// TIA Portal project "PTAR" (V16)

(* hardware
DEVICE "S7-1200 station_1"  S7-1200 Station
   slot 0: "Rack_0"  S7-1200 Rack  Rack  V1.0
   slot 1: "PLC_1 Agua de servicio"  CPU 1214C DC/DC/Rly  6ES7 214-1HG40-0XB0  V4.4
   slot 2: "DI 16x24VDC/DQ 16xRelay_1"  SM 1223 DI16/DQ16 x relay  6ES7 223-1PL32-0XB0  V2.0
   slot 3: "DI 16x24VDC_1"  6ES7 221-1BH32-0XB0  V2.0
   slot 4: "DI 16x24VDC_2"  6ES7 221-1BH32-0XB0  V2.0
   slot 5: "DI 16x24VDC_3"  6ES7 221-1BH32-0XB0  V2.0
   slot 6: "AI 8x13BIT_1"  6ES7 231-4HF32-0XB0  V2.1
   slot 7: "AI 8x13BIT_2"  6ES7 231-4HF32-0XB0  V2.1
   slot 101: "CM 1241 (RS422/485)_1"  6ES7 241-1CH32-0XB0  V2.2
DEVICE "S7-1200 station_2"  S7-1200 Station
   slot 0: "Rack_0"  S7-1200 Rack  Rack  V1.0
   slot 1: "PLC_2 Compresores y agua potable"  CPU 1214C AC/DC/Rly  6ES7 214-1BG40-0XB0  V4.4
   slot 2: "DI 16x24VDC/DQ 16xRelay_1"  6ES7 223-1BL32-0XB0  V2.0
   slot 3: "DI 16x24VDC/DQ 16xRelay_2"  SM 1223 DI16/DQ16 x relay  6ES7 223-1PL32-0XB0  V2.0
   slot 4: "DI 16x24VDC_1"  6ES7 221-1BH32-0XB0  V2.0
   slot 5: "DI 16x24VDC_2"  6ES7 221-1BH32-0XB0  V2.0
   slot 6: "AI 8x13BIT_1"  6ES7 231-4HF32-0XB0  V2.1
   slot 7: "AI 8x13BIT_2"  6ES7 231-4HF32-0XB0  V2.1
   slot 101: "CM 1241 (RS422/485)_1"  6ES7 241-1CH32-0XB0  V2.2
*)

// ===== PLC "PLC_1 Agua de servicio"  CPU 1214C DC/DC/Rly =====

VAR_GLOBAL   // PLC tag table "Tabla de variables estándar"
   "PARO EMERGENCIA TAB AGUA SERVICIO LOCAL" AT %I0.0 : Bool;
   "FALLA BREAKER TOTALIZADOR" AT %I0.1 : Bool;
   "FALLA BREAKER BOMBA 096P001A" AT %I0.2 : Bool;
   "FALLA BREAKER BOMBA 096P001B" AT %I0.3 : Bool;
   "FALLA BREAKER BOMBA 096P001C" AT %I0.4 : Bool;
   "FALLA BREAKER BOMBA 096P001D" AT %I0.5 : Bool;
   "FALLA BREAKER BOMBA 096P001E" AT %I0.6 : Bool;
   "FALLA BREAKER BOMBA 096P001F" AT %I0.7 : Bool;
   "SELEC TAB MODO CCM BOMBA 096P001A" AT %I1.0 : Bool;
   "SELEC TAB MODO CAMPO BOMBA 096P001A" AT %I1.1 : Bool;
   "SELEC TAB MODO REMOTO BOMBA 096P001A" AT %I1.2 : Bool;
   "SELEC TAB MODO CCM BOMBA 096P001B" AT %I1.3 : Bool;
   "SELEC TAB MODO CAMPO BOMBA 096P001B" AT %I1.4 : Bool;
   "SELEC TAB MODO REMOTO BOMBA 096P001B" AT %I1.5 : Bool;
   "SELEC TAB MODO CCM BOMBA 096P001C" AT %I2.0 : Bool;
   "SELEC TAB MODO CAMPO BOMBA 096P001C" AT %I2.1 : Bool;
   "SELEC TAB MODO REMOTO BOMBA 096P001C" AT %I2.2 : Bool;
   "SELEC TAB MODO CCM BOMBA 096P001D" AT %I2.3 : Bool;
   "SELEC TAB MODO CAMPO BOMBA 096P001D" AT %I2.4 : Bool;
   "SELEC TAB MODO REMOTO BOMBA 096P001D" AT %I2.5 : Bool;
   "SELEC TAB MODO CCM BOMBA 096P001E" AT %I2.6 : Bool;
   "SELEC TAB MODO CAMPO BOMBA 096P001E" AT %I2.7 : Bool;
   "SELEC TAB MODO REMOTO BOMBA 096P001E" AT %I3.0 : Bool;
   "SELEC TAB MODO CCM BOMBA 096P001F" AT %I3.1 : Bool;
   "SELEC TAB MODO CAMPO BOMBA 096P001F" AT %I3.2 : Bool;
   "SELEC TAB MODO REMOTO BOMBA 096P001F" AT %I3.3 : Bool;
   "PULSADOR START CCM 096P001A" AT %I3.4 : Bool;
   "PULSADOR STOP CCM 096P001A" AT %I3.5 : Bool;
   "PULSADOR START CCM 096P001B" AT %I3.6 : Bool;
   "PULSADOR STOP CCM 096P001B" AT %I3.7 : Bool;
   "PULSADOR START CCM 096P001C" AT %I4.0 : Bool;
   "PULSADOR STOP CCM 096P001C" AT %I4.1 : Bool;
   "PULSADOR START CCM 096P001D" AT %I4.2 : Bool;
   "PULSADOR STOP CCM 096P001D" AT %I4.3 : Bool;
   "PULSADOR START CCM 096P001E" AT %I4.4 : Bool;
   "PULSADOR STOP CCM 096P001E" AT %I4.5 : Bool;
   "PULSADOR START CCM 096P001F" AT %I4.6 : Bool;
   "PULSADOR STOP CCM 096P001F" AT %I4.7 : Bool;
   "PULSADOR RESET CCM 096P001A" AT %I5.0 : Bool;
   "PULSADOR RESET CCM 096P001B" AT %I5.1 : Bool;
   "PULSADOR RESET CCM 096P001C" AT %I5.2 : Bool;
   "PULSADOR RESET CCM 096P001D" AT %I5.3 : Bool;
   "PULSADOR RESET CCM 096P001E" AT %I5.4 : Bool;
   "PULSADOR RESET CCM 096P001F" AT %I5.5 : Bool;
   "PARO EMERGENCIA 096P001A CAMPO" AT %I7.5 : Bool;
   "PULSADOR START CAMPO 096P001A" AT %I5.7 : Bool;
   "PULSADOR STOP CAMPO 096P001A" AT %I6.0 : Bool;
   "PULSADOR START CAMPO 096P001B" AT %I6.1 : Bool;
   "PULSADOR STOP CAMPO 096P001B" AT %I6.2 : Bool;
   "PULSADOR START CAMPO 096P001C" AT %I6.3 : Bool;
   "PULSADOR STOP CAMPO 096P001C" AT %I6.4 : Bool;
   "PULSADOR START CAMPO 096P001D" AT %I6.5 : Bool;
   "PULSADOR STOP CAMPO 096P001D" AT %I6.6 : Bool;
   "PULSADOR START CAMPO 096P001E" AT %I6.7 : Bool;
   "PULSADOR STOP CAMPO 096P001E" AT %I7.0 : Bool;
   "PULSADOR START CAMPO 096P001F" AT %I7.1 : Bool;
   "PULSADOR STOP CAMPO 096P001F" AT %I7.2 : Bool;
   "SWITCH DE BAJA PRESION AGUA DE SERVICIO" AT %I7.3 : Bool;
   "SWITCH DE FLUJO AGUA DE SERVICIO" AT %I7.4 : Bool;
   "TRANSMISOR DE PRESION EN SUCCION 096PIT001" AT %IW300 : Word;
   "TRANSMISOR DE PRESION EN DESCARGA 096PIT002" AT %IW302 : Word;
   "PARO EMERGENCIA 096P001B CAMPO" AT %I7.6 : Bool;
   "PARO EMERGENCIA 096P001C CAMPO" AT %I7.7 : Bool;
   "PARO EMERGENCIA 096P001D CAMPO" AT %I8.0 : Bool;
   "PARO EMERGENCIA 096P001E CAMPO" AT %I8.1 : Bool;
   "PARO EMERGENCIA 096P001F CAMPO" AT %I8.2 : Bool;
   "PERMISO DE ARRANQUE" AT %I8.3 : Bool;
   "ENTRADAS DIGITALES GRUPO 1" AT %IW0 : Word;
   "ENTRADAS DIGITALES GRUPO 2" AT %IW2 : Word;
   "ENTRADAS DIGITALES GRUPO 3" AT %IW7 : Word;
   "Tag_1" AT %I8.4 : Bool;
   "OPERANDO BOMBA 096P001A" AT %Q0.0 : Bool;
   "FALLA BOMBA 096P001A" AT %Q0.1 : Bool;
   "OPERANDO BOMBA 096P001B" AT %Q0.2 : Bool;
   "FALLA BOMBA 096P001B" AT %Q0.3 : Bool;
   "OPERANDO BOMBA 096P001C" AT %Q0.4 : Bool;
   "FALLA BOMBA 096P001C" AT %Q0.5 : Bool;
   "OPERANDO BOMBA 096P001D" AT %Q0.6 : Bool;
   "FALLA BOMBA 096P001D" AT %Q0.7 : Bool;
   "OPERANDO BOMBA 096P001E" AT %Q1.0 : Bool;
   "FALLA BOMBA 096P001E" AT %Q1.1 : Bool;
   "OPERANDO BOMBA 096P001F" AT %Q2.0 : Bool;
   "FALLA BOMBA 096P001F" AT %Q2.1 : Bool;
   "SALIDAS DIGITALES GRUPO 1" AT %QW0 : Word;
   "CONSIGNA FRECUENCIA AGUA RESIDUAL" AT %MD100 : Real;
   "SLEEP BOOSTER" AT %M10.0 : Bool;
   "INICIAR BOMBA" AT %M10.1 : Bool;
   "Clock_Byte" AT %MB0 : Byte;
   "Clock_10Hz" AT %M0.0 : Bool;
   "Clock_5Hz" AT %M0.1 : Bool;
   "Clock_2.5Hz" AT %M0.2 : Bool;
   "Clock_2Hz" AT %M0.3 : Bool;
   "Clock_1.25Hz" AT %M0.4 : Bool;
   "Clock_1Hz" AT %M0.5 : Bool;
   "Clock_0.625Hz" AT %M0.6 : Bool;
   "Clock_0.5Hz" AT %M0.7 : Bool;
   "System_Byte" AT %MB1 : Byte;
   "FirstScan" AT %M1.0 : Bool;
   "DiagStatusUpdate" AT %M1.1 : Bool;
   "AlwaysTRUE" AT %M1.2 : Bool;
   "AlwaysFALSE" AT %M1.3 : Bool;
   "DISPONIBLE BOMBA A" AT %M10.2 : Bool;
   "DISPONIBLE BOMBA B" AT %M10.3 : Bool;
   "DISPONIBLE BOMBA C" AT %M10.4 : Bool;
   "DISPONIBLE BOMBA D" AT %M10.5 : Bool;
   "DISPONIBLE BOMBA E" AT %M10.6 : Bool;
   "DISPONIBLE BOMBA F" AT %M10.7 : Bool;
   "BOMBA LIDER 1" AT %M11.0 : Bool;
   "BOMBA LIDER 2" AT %M11.1 : Bool;
   "BOMBA LIDER 3" AT %M11.2 : Bool;
   "BOMBA LIDER 4" AT %M11.3 : Bool;
   "BOMBA LIDER 5" AT %M11.4 : Bool;
   "BOMBA LIDER 6" AT %M11.5 : Bool;
   "AD1" AT %M12.0 : Bool;
   "HABILITACION SISTEMA" AT %M12.1 : Bool;
   "AD2" AT %M12.2 : Bool;
   "AD3" AT %M12.3 : Bool;
   "AD4" AT %M12.4 : Bool;
   "AD5" AT %M12.5 : Bool;
   "ARRANQUE BOMBA A" AT %M13.0 : Bool;
   "ARRANQUE BOMBA B" AT %M13.1 : Bool;
   "ARRANQUE BOMBA C" AT %M13.2 : Bool;
   "ARRANQUE BOMBA D" AT %M13.4 : Bool;
   "ARRANQUE BOMBA E" AT %M13.5 : Bool;
   "ARRANQUE BOMBA F" AT %M13.6 : Bool;
   "PRESION OK" AT %M13.7 : Bool;
   "Tag_3" AT %M14.0 : Bool;
   "Tag_4" AT %M14.1 : Bool;
   "Tag_5" AT %M14.2 : Bool;
   "Tag_6" AT %M14.3 : Bool;
   "Tag_7" AT %M14.4 : Bool;
   "Tag_8" AT %M14.5 : Bool;
   "Tag_9" AT %M14.6 : Bool;
   "Tag_10" AT %M14.7 : Bool;
   "Tag_11" AT %M15.0 : Bool;
   "Tag_12" AT %M15.1 : Bool;
   "Tag_13" AT %M15.2 : Bool;
   "Tag_14" AT %M15.3 : Bool;
   "RESET GENERAL" AT %M2.0 : Bool;
   "ALARMA GENERAL" AT %M2.1 : Bool;
   "Tag_2" AT %M16.0 : Bool;
   "Tag_15" AT %M16.1 : Bool;
   "Tag_16" AT %M16.2 : Bool;
   "Tag_17" AT %M16.3 : Bool;
   "Tag_18" AT %M16.4 : Bool;
   "Tag_19" AT %M16.5 : Bool;
   "Tag_20" AT %M16.6 : Bool;
   "Tag_21" AT %M16.7 : Bool;
   "Tag_22" AT %M17.0 : Bool;
   "Tag_23" AT %M17.1 : Bool;
   "Tag_24" AT %M17.2 : Bool;
   "Tag_25" AT %M17.3 : Bool;
   "Tag_26" AT %M17.4 : Bool;
   "Tag_27" AT %M17.5 : Bool;
   "Tag_28" AT %M17.6 : Bool;
   "Tag_29" AT %M17.7 : Bool;
   "Tag_30" AT %M18.0 : Bool;
   "Tag_31" AT %M18.1 : Bool;
END_VAR

DATA_BLOCK "ANALOGAS"   // DB1
{ S7_Optimized_Access := 'TRUE' }
VERSION : 0.1
   VAR RETAIN
      "096PIT001" : Struct
         "CD MAX" : DInt := 27648;
         "CD MIN" : DInt := 0;
         "ING MAX" : Real := 232.0;
         "ING MIN" : Real := 0.0;
         HH : Real := 50.0;
         H : Real := 15.0;
         L : Real := 2.0;
         LL : Real := 1.5;
         ESCALIZADA : Real := 3.608217;
         PORCENTAJE : Real := 1.555266;
      END_STRUCT;
      "096PIT002" : Struct
         "CD MAX" : DInt := 27648;
         "CD MIN" : DInt := 0;
         "ING MAX" : Real := 232.0;
         "ING MIN" : Real := 0.0;
         HH : Real := 120.0;
         H : Real := 100.0;
         L : Real := 30.0;
         LL : Real := 20.0;
         ESCALIZADA : Real := 67.6331;
         PORCENTAJE : Real := 29.1522;
      END_STRUCT;
   END_VAR
BEGIN
END_DATA_BLOCK

DATA_BLOCK "BOTONERA"   // DB2
{ S7_Optimized_Access := 'TRUE' }
VERSION : 0.1
   VAR
      "096P001A" : Struct
         START : Bool;
         STOP : Bool;
         FALLA : Bool;
         "RESET FALLA" : Bool;
         "RESET TIEMPO OPERANDO" : Bool;
         "RESET TIEMPO ACUMULADO" : Bool;
      END_STRUCT;
      "096P001B" : Struct
         START : Bool;
         STOP : Bool;
         FALLA : Bool;
         "RESET FALLA" : Bool;
         "RESET TIEMPO OPERANDO" : Bool;
         "RESET TIEMPO ACUMULADO" : Bool;
      END_STRUCT;
      "096P001C" : Struct
         START : Bool;
         STOP : Bool;
         FALLA : Bool;
         "RESET FALLA" : Bool;
         "RESET TIEMPO OPERANDO" : Bool;
         "RESET TIEMPO ACUMULADO" : Bool;
      END_STRUCT;
      "096P001D" : Struct
         START : Bool;
         STOP : Bool;
         FALLA : Bool;
         "RESET FALLA" : Bool;
         "RESET TIEMPO OPERANDO" : Bool;
         "RESET TIEMPO ACUMULADO" : Bool;
      END_STRUCT;
      "096P001E" : Struct
         START : Bool;
         STOP : Bool;
         FALLA : Bool;
         "RESET FALLA" : Bool;
         "RESET TIEMPO OPERANDO" : Bool;
         "RESET TIEMPO ACUMULADO" : Bool;
      END_STRUCT;
      "096P001F" : Struct
         START : Bool;
         STOP : Bool;
         FALLA : Bool;
         "RESET FALLA" : Bool;
         "RESET TIEMPO OPERANDO" : Bool;
         "RESET TIEMPO ACUMULADO" : Bool;
      END_STRUCT;
      "TODO A MANUAL" : Bool;
      "TODO A AUTOMATICO" : Bool;
      "TODO EN MANUAL" : Bool;
      "TODO EN AUTOMATICO" : Bool;
   END_VAR
BEGIN
END_DATA_BLOCK

DATA_BLOCK "MODO OPERACION"   // DB3
{ S7_Optimized_Access := 'TRUE' }
VERSION : 0.1
   VAR RETAIN
      "096P001A" : Struct
         MANUAL : Bool;
         AUTOMATICO : Bool;
         SCADA : Bool;
      END_STRUCT;
      "096P001B" : Struct
         MANUAL : Bool;
         AUTOMATICO : Bool;
         SCADA : Bool;
      END_STRUCT;
      "096P001C" : Struct
         MANUAL : Bool;
         AUTOMATICO : Bool;
         SCADA : Bool;
      END_STRUCT;
      "096P001D" : Struct
         MANUAL : Bool;
         AUTOMATICO : Bool;
         SCADA : Bool;
      END_STRUCT;
      "096P001E" : Struct
         MANUAL : Bool;
         AUTOMATICO : Bool;
         SCADA : Bool;
      END_STRUCT;
      "096P001F" : Struct
         MANUAL : Bool;
         AUTOMATICO : Bool;
         SCADA : Bool;
      END_STRUCT;
   END_VAR
BEGIN
END_DATA_BLOCK

DATA_BLOCK "ESC HZ"   // DB4
{ S7_Optimized_Access := 'TRUE' }
VERSION : 0.1
   VAR RETAIN
      "096P001A" : Struct
         "FRECUENCIA MAX" : Real := 60.0;
         "FRECUENCIA MIN" : Real := 20.0;
         "FRECUENCIA OP" : Real := 60.0;
      END_STRUCT;
      "096P001B" : Struct
         "FRECUENCIA MAX" : Real := 60.0;
         "FRECUENCIA MIN" : Real := 20.0;
         "FRECUENCIA OP" : Real := 60.0;
      END_STRUCT;
      "096P001C" : Struct
         "FRECUENCIA MAX" : Real := 60.0;
         "FRECUENCIA MIN" : Real := 20.0;
         "FRECUENCIA OP" : Real := 60.0;
      END_STRUCT;
      "096P001D" : Struct
         "FRECUENCIA MAX" : Real := 60.0;
         "FRECUENCIA MIN" : Real := 20.0;
         "FRECUENCIA OP" : Real := 60.0;
      END_STRUCT;
      "096P001E" : Struct
         "FRECUENCIA MAX" : Real := 60.0;
         "FRECUENCIA MIN" : Real := 20.0;
         "FRECUENCIA OP" : Real := 60.0;
      END_STRUCT;
      "096P001F" : Struct
         "FRECUENCIA MAX" : Real := 60.0;
         "FRECUENCIA MIN" : Real := 20.0;
         "FRECUENCIA OP" : Real := 60.0;
      END_STRUCT;
   END_VAR
BEGIN
END_DATA_BLOCK

DATA_BLOCK "DATOS LECTURA VFDS"   // DB5
{ S7_Optimized_Access := 'TRUE' }
VERSION : 0.1
   VAR
      "096P001A" : Struct
         AMPERAJE : Real;
         FRECUENCIA : Real;
         "FRECUENCIA %" : Real;
         VOLTAJE : Real;
         ESTADO : Bool;
      END_STRUCT;
      "096P001B" : Struct
         AMPERAJE : Real;
         FRECUENCIA : Real;
         "FRECUENCIA %" : Real;
         VOLTAJE : Real;
         ESTADO : Bool;
      END_STRUCT;
      "096P001C" : Struct
         AMPERAJE : Real;
         FRECUENCIA : Real;
         "FRECUENCIA %" : Real;
         VOLTAJE : Real;
         ESTADO : Bool;
      END_STRUCT;
      "096P001D" : Struct
         AMPERAJE : Real;
         FRECUENCIA : Real;
         "FRECUENCIA %" : Real;
         VOLTAJE : Real;
         ESTADO : Bool;
      END_STRUCT;
      "096P001E" : Struct
         AMPERAJE : Real;
         FRECUENCIA : Real;
         "FRECUENCIA %" : Real;
         VOLTAJE : Real;
         ESTADO : Bool;
      END_STRUCT;
      "096P001F" : Struct
         AMPERAJE : Real;
         FRECUENCIA : Real;
         "FRECUENCIA %" : Real;
         VOLTAJE : Real;
         ESTADO : Bool;
      END_STRUCT;
   END_VAR
BEGIN
END_DATA_BLOCK

DATA_BLOCK "CONFIG SIS PRESION AGUA SERVICIO"   // DB25
{ S7_Optimized_Access := 'TRUE' }
VERSION : 0.1
   VAR RETAIN
      "DESVIO DE PRESION PARA DESPERTAR" : Real := 10.0;
      "VALOR DE FRECUENCIA PARA DORMIR" : Real := 40.0;
      "TIEMPO PARA MODO DORMIR" : Real := 40.0;
      "FRECUENCIA PARA ARRANCAR BOMBA EN PARALELO" : Real := 59.0;
      "TIEMPO PARA ARRANCAR BOMBA EN PARALELO" : Real := 40.0;
      "FRECUENCIA PARA APAGAR BOMBA EN PARALELO" : Real := 43.0;
      "TIEMPO PARA APAGAR BOMBA EN PARALELO" : Real := 5.0;
      "TORQUE MINIMO PARA DETECCION BOMBA EN VACIO" : Real := 20.0;
      "TIEMPO DETECCION BOMBA EN VACIO" : Real := 10.0;
      "PRESION BOOSTER" : Real := 2.0;
      "TIEMPO SLEEP BOOSTER" : Real := 10.0;
      "FRECUENCIA MAXIMA CONFIGURADA EN VFDS" : Real := 60.0;
      "FRECUENCIA MINIMA CONFIGURADA EN VFDS" : Real := 37.0;
      "TIEMPO DE ALTERNACION" : Int := 10;
      SETPOINT : Real := 80.0;
      "SETPOINT %" : Real := 34.61207;
      K : Real := 0.0;
      TI : Real := 0.0;
      TD : Real := 0.0;
   END_VAR
   VAR
      "SALIDA PID %" : Real := 0.0;
   END_VAR
BEGIN
END_DATA_BLOCK

DATA_BLOCK "DATOS ESCRITURA VFDS"   // DB30
{ S7_Optimized_Access := 'TRUE' }
VERSION : 0.1
   VAR
      "096P001A" : Struct
         FRECUENCIA : Real;
      END_STRUCT;
      "096P001B" : Struct
         FRECUENCIA : Real;
      END_STRUCT;
      "096P001C" : Struct
         FRECUENCIA : Real;
      END_STRUCT;
      "096P001D" : Struct
         FRECUENCIA : Real;
      END_STRUCT;
      "096P001E" : Struct
         FRECUENCIA : Real;
      END_STRUCT;
      "096P001F" : Struct
         FRECUENCIA : Real;
      END_STRUCT;
   END_VAR
BEGIN
END_DATA_BLOCK

DATA_BLOCK "Alarmas Sis servicio"   // DB37
{ S7_Optimized_Access := 'TRUE' }
VERSION : 0.1
   VAR
      "Alarma general" : Bool;
      "Reset alarmas" : Bool;
   END_VAR
BEGIN
END_DATA_BLOCK

DATA_BLOCK "LECTURA VFD1"   // DB40
{ S7_Optimized_Access := 'FALSE' }
VERSION : 0.1
   VAR
      "40007+" : Array[0..8] of Int;
      "40016+" : Array[0..7] of Int;
      "40816+" : Array[0..1] of Int;
   END_VAR
BEGIN
END_DATA_BLOCK

DATA_BLOCK "LECTURA VFD2"   // DB41
{ S7_Optimized_Access := 'FALSE' }
VERSION : 0.1
   VAR
      "40007+" : Array[0..8] of Int;
      "40016+" : Array[0..7] of Int;
      "40816+" : Array[0..1] of Int;
   END_VAR
BEGIN
END_DATA_BLOCK

DATA_BLOCK "LECTURA VFD3"   // DB42
{ S7_Optimized_Access := 'FALSE' }
VERSION : 0.1
   VAR
      "40007+" : Array[0..8] of Int;
      "40016+" : Array[0..7] of Int;
      "40816+" : Array[0..1] of Int;
   END_VAR
BEGIN
END_DATA_BLOCK

DATA_BLOCK "LECTURA VFD4"   // DB43
{ S7_Optimized_Access := 'FALSE' }
VERSION : 0.1
   VAR
      "40007+" : Array[0..8] of Int;
      "40016+" : Array[0..7] of Int;
      "40816+" : Array[0..1] of Int;
   END_VAR
BEGIN
END_DATA_BLOCK

DATA_BLOCK "LECTURA VFD5"   // DB44
{ S7_Optimized_Access := 'FALSE' }
VERSION : 0.1
   VAR
      "40007+" : Array[0..8] of Int;
      "40016+" : Array[0..7] of Int;
      "40816+" : Array[0..1] of Int;
   END_VAR
BEGIN
END_DATA_BLOCK

DATA_BLOCK "LECTURA VFD6"   // DB45
{ S7_Optimized_Access := 'FALSE' }
VERSION : 0.1
   VAR
      "40007+" : Array[0..8] of Int;
      "40016+" : Array[0..7] of Int;
      "40816+" : Array[0..1] of Int;
   END_VAR
BEGIN
END_DATA_BLOCK

DATA_BLOCK "ESCRITURA VFD1"   // DB47
{ S7_Optimized_Access := 'FALSE' }
VERSION : 0.1
   VAR
      "40005+" : Array[0..1] of Int;
   END_VAR
BEGIN
END_DATA_BLOCK

DATA_BLOCK "ESCRITURA VFD2"   // DB48
{ S7_Optimized_Access := 'FALSE' }
VERSION : 0.1
   VAR
      "40005+" : Array[0..1] of Int;
   END_VAR
BEGIN
END_DATA_BLOCK

DATA_BLOCK "ESCRITURA VFD3"   // DB49
{ S7_Optimized_Access := 'FALSE' }
VERSION : 0.1
   VAR
      "40005+" : Array[0..1] of Int;
   END_VAR
BEGIN
END_DATA_BLOCK

DATA_BLOCK "ESCRITURA VFD4"   // DB50
{ S7_Optimized_Access := 'FALSE' }
VERSION : 0.1
   VAR
      "40005+" : Array[0..1] of Int;
   END_VAR
BEGIN
END_DATA_BLOCK

DATA_BLOCK "ESCRITURA VFD5"   // DB51
{ S7_Optimized_Access := 'FALSE' }
VERSION : 0.1
   VAR
      "40005+" : Array[0..1] of Int;
   END_VAR
BEGIN
END_DATA_BLOCK

DATA_BLOCK "ESCRITURA VFD6"   // DB52
{ S7_Optimized_Access := 'FALSE' }
VERSION : 0.1
   VAR
      "40005+" : Array[0..1] of Int;
   END_VAR
BEGIN
END_DATA_BLOCK

DATA_BLOCK "DATA MODBUS TCP"   // DB78
{ S7_Optimized_Access := 'FALSE' }
VERSION : 0.1
   VAR
      DATA : Array[0..100] of Word;
   END_VAR
BEGIN
END_DATA_BLOCK

DATA_BLOCK "MB CONFIG"   // DB79
{ S7_Optimized_Access := 'FALSE' }
VERSION : 0.1
   VAR
      CONNECT : TCON_IP_v4;
      NDR : Bool;
      DR : Bool;
      ERROR : Bool;
      STATUS : Word;
   END_VAR
BEGIN
   CONNECT.InterfaceId := 64;
   CONNECT.ID := 1;
   CONNECT.ConnectionType := 11;
   CONNECT.LocalPort := 502;
END_DATA_BLOCK

DATA_BLOCK "FALLAS HMI"   // DB93
{ S7_Optimized_Access := 'FALSE' }
VERSION : 0.1
   VAR
      "PARO EMERGENCIA ACTIVO SISTEMA GRAL AGUA SERVICIO" : Bool;
      "FALLA BREAKER PRINCIPAL" : Bool;
      "FALLA BREAKER Q1 - VFD 1 096P001A" : Bool;
      "FALLA VARIADOR VELOCIDAD 096P001A" : Bool;
      "PARO DE EMERGENCIA ACTIVO 096P001A" : Bool;
      "NO CONFIRMA ARRANQUE BOMBA 096P001A" : Bool;
      "FALLA BREAKER Q2 - VFD 2 096P001B" : Bool;
      "FALLA VARIADOR VELOCIDAD 096P001B" : Bool;
      "PARO DE EMERGENCIA ACTIVO 096P001B" : Bool;
      "NO CONFIRMA ARRANQUE BOMBA 096P001B" : Bool;
      "FALLA BREAKER Q3 - VFD 3 096P001C" : Bool;
      "FALLA VARIADOR VELOCIDAD 096P001C" : Bool;
      "PARO DE EMERGENCIA ACTIVO 096P001C" : Bool;
      "NO CONFIRMA ARRANQUE BOMBA 096P001C" : Bool;
      "FALLA BREAKER Q4 - VFD 4 096P001D" : Bool;
      "FALLA VARIADOR VELOCIDAD 096P001D" : Bool;
      "PARO DE EMERGENCIA ACTIVO 096P001D" : Bool;
      "NO CONFIRMA ARRANQUE BOMBA 096P001D" : Bool;
      "FALLA BREAKER Q5 - VFD 5 096P001E" : Bool;
      "FALLA VARIADOR VELOCIDAD 096P001E" : Bool;
      "PARO DE EMERGENCIA ACTIVO 096P001E" : Bool;
      "NO CONFIRMA ARRANQUE BOMBA 096P001E" : Bool;
      "FALLA BREAKER Q6 - VFD 6 096P001F" : Bool;
      "FALLA VARIADOR VELOCIDAD 096P001F" : Bool;
      "PARO DE EMERGENCIA ACTIVO 096P001F" : Bool;
      "NO CONFIRMA ARRANQUE BOMBA 096P001F" : Bool;
      "SWITCH DE FLUJO EN SUCCION INACTIVO FSL001" : Bool;
      "SWITCH DE PRESION EN SUCCION INACTIVO PSL001" : Bool;
      "NO CONFIRMA SWITCH DE FLUJO CON BOMBA 096P001A" : Bool;
      "NO CONFIRMA SWITCH DE FLUJO CON BOMBA 096P001B" : Bool;
      "NO CONFIRMA SWITCH DE FLUJO CON BOMBA 096P001C" : Bool;
      "NO CONFIRMA SWITCH DE FLUJO CON BOMBA 096P001D" : Bool;
      "NO CONFIRMA SWITCH DE FLUJO CON BOMBA 096P001E" : Bool;
      "NO CONFIRMA SWITCH DE FLUJO CON BOMBA 096P001F" : Bool;
      "FALLA POR ALTA PRESION DE DESCARGA 096PIT002" : Bool;
      "ALARMA POR ALTA PRESION DE DESCARGA 096PIT002" : Bool;
      "ALARMA POR BAJA PRESION DE DESCARGA 096PIT002" : Bool;
      "FALLA POR BAJA PRESION DE DESCARGA 096PIT002" : Bool;
      "FALLA POR ALTA PRESION DE SUCCION 096PIT001" : Bool;
      "ALARMA POR ALTA PRESION DE SUCCION 096PIT001" : Bool;
      "ALARMA POR BAJA PRESION DE SUCCION 096PIT001" : Bool;
      "FALLA POR BAJA PRESION DE SUCCION 096PIT001" : Bool;
   END_VAR
BEGIN
END_DATA_BLOCK

// folder: System blocks/Program resources

DATA_BLOCK "TEMPO MODO MANUAL 001A"   // DB6
{ S7_Optimized_Access := 'TRUE' }
AUTHOR : Simatic
FAMILY : IEC
NAME : IEC_TMR
VERSION : 1.0
// stored: InstanceOfName IEC_TIMER
"IEC_TIMER"
BEGIN
END_DATA_BLOCK

DATA_BLOCK "TEMPO MODO AUTOMATICO 001A"   // DB7
{ S7_Optimized_Access := 'TRUE' }
AUTHOR : Simatic
FAMILY : IEC
NAME : IEC_TMR
VERSION : 1.0
// stored: InstanceOfName IEC_TIMER
"IEC_TIMER"
BEGIN
END_DATA_BLOCK

DATA_BLOCK "TEMPO MODO SCADA 001A"   // DB8
{ S7_Optimized_Access := 'TRUE' }
AUTHOR : Simatic
FAMILY : IEC
NAME : IEC_TMR
VERSION : 1.0
// stored: InstanceOfName IEC_TIMER
"IEC_TIMER"
BEGIN
END_DATA_BLOCK

DATA_BLOCK "TEMPO MODO MANUAL 001B"   // DB9
{ S7_Optimized_Access := 'TRUE' }
AUTHOR : Simatic
FAMILY : IEC
NAME : IEC_TMR
VERSION : 1.0
// stored: InstanceOfName IEC_TIMER
"IEC_TIMER"
BEGIN
END_DATA_BLOCK

DATA_BLOCK "TEMPO MODO AUTOMATICO 001B"   // DB10
{ S7_Optimized_Access := 'TRUE' }
AUTHOR : Simatic
FAMILY : IEC
NAME : IEC_TMR
VERSION : 1.0
// stored: InstanceOfName IEC_TIMER
"IEC_TIMER"
BEGIN
END_DATA_BLOCK

DATA_BLOCK "TEMPO MODO SCADA 001B"   // DB11
{ S7_Optimized_Access := 'TRUE' }
AUTHOR : Simatic
FAMILY : IEC
NAME : IEC_TMR
VERSION : 1.0
// stored: InstanceOfName IEC_TIMER
"IEC_TIMER"
BEGIN
END_DATA_BLOCK

DATA_BLOCK "TEMPO MODO MANUAL 001C"   // DB12
{ S7_Optimized_Access := 'TRUE' }
AUTHOR : Simatic
FAMILY : IEC
NAME : IEC_TMR
VERSION : 1.0
// stored: InstanceOfName IEC_TIMER
"IEC_TIMER"
BEGIN
END_DATA_BLOCK

DATA_BLOCK "TEMPO MODO AUTOMATICO 001C"   // DB13
{ S7_Optimized_Access := 'TRUE' }
AUTHOR : Simatic
FAMILY : IEC
NAME : IEC_TMR
VERSION : 1.0
// stored: InstanceOfName IEC_TIMER
"IEC_TIMER"
BEGIN
END_DATA_BLOCK

DATA_BLOCK "TEMPO MODO SCADA 001C"   // DB14
{ S7_Optimized_Access := 'TRUE' }
AUTHOR : Simatic
FAMILY : IEC
NAME : IEC_TMR
VERSION : 1.0
// stored: InstanceOfName IEC_TIMER
"IEC_TIMER"
BEGIN
END_DATA_BLOCK

DATA_BLOCK "TEMPO MODO MANUAL 001D"   // DB15
{ S7_Optimized_Access := 'TRUE' }
AUTHOR : Simatic
FAMILY : IEC
NAME : IEC_TMR
VERSION : 1.0
// stored: InstanceOfName IEC_TIMER
"IEC_TIMER"
BEGIN
END_DATA_BLOCK

DATA_BLOCK "TEMPO MODO AUTOMATICO 001D"   // DB16
{ S7_Optimized_Access := 'TRUE' }
AUTHOR : Simatic
FAMILY : IEC
NAME : IEC_TMR
VERSION : 1.0
// stored: InstanceOfName IEC_TIMER
"IEC_TIMER"
BEGIN
END_DATA_BLOCK

DATA_BLOCK "TEMPO MODO SCADA 001D"   // DB17
{ S7_Optimized_Access := 'TRUE' }
AUTHOR : Simatic
FAMILY : IEC
NAME : IEC_TMR
VERSION : 1.0
// stored: InstanceOfName IEC_TIMER
"IEC_TIMER"
BEGIN
END_DATA_BLOCK

DATA_BLOCK "TEMPO MODO MANUAL 001E"   // DB18
{ S7_Optimized_Access := 'TRUE' }
AUTHOR : Simatic
FAMILY : IEC
NAME : IEC_TMR
VERSION : 1.0
// stored: InstanceOfName IEC_TIMER
"IEC_TIMER"
BEGIN
END_DATA_BLOCK

DATA_BLOCK "TEMPO MODO AUTOMATICO 001E"   // DB19
{ S7_Optimized_Access := 'TRUE' }
AUTHOR : Simatic
FAMILY : IEC
NAME : IEC_TMR
VERSION : 1.0
// stored: InstanceOfName IEC_TIMER
"IEC_TIMER"
BEGIN
END_DATA_BLOCK

DATA_BLOCK "TEMPO MODO SCADA 001E"   // DB20
{ S7_Optimized_Access := 'TRUE' }
AUTHOR : Simatic
FAMILY : IEC
NAME : IEC_TMR
VERSION : 1.0
// stored: InstanceOfName IEC_TIMER
"IEC_TIMER"
BEGIN
END_DATA_BLOCK

DATA_BLOCK "TEMPO MODO SCADA 001F"   // DB21
{ S7_Optimized_Access := 'TRUE' }
AUTHOR : Simatic
FAMILY : IEC
NAME : IEC_TMR
VERSION : 1.0
// stored: InstanceOfName IEC_TIMER
"IEC_TIMER"
BEGIN
END_DATA_BLOCK

DATA_BLOCK "TEMPO MODO AUTOMATICO 001F"   // DB22
{ S7_Optimized_Access := 'TRUE' }
AUTHOR : Simatic
FAMILY : IEC
NAME : IEC_TMR
VERSION : 1.0
// stored: InstanceOfName IEC_TIMER
"IEC_TIMER"
BEGIN
END_DATA_BLOCK

DATA_BLOCK "TEMPO MODO MANUAL 001F"   // DB23
{ S7_Optimized_Access := 'TRUE' }
AUTHOR : Simatic
FAMILY : IEC
NAME : IEC_TMR
VERSION : 1.0
// stored: InstanceOfName IEC_TIMER
"IEC_TIMER"
BEGIN
END_DATA_BLOCK

DATA_BLOCK "TIEMPO PARA APAGAR"   // DB26
{ S7_Optimized_Access := 'TRUE' }
AUTHOR : Simatic
FAMILY : IEC
NAME : IEC_TMR
VERSION : 1.0
// stored: InstanceOfName IEC_TIMER
"IEC_TIMER"
BEGIN
END_DATA_BLOCK

DATA_BLOCK "TIEMPO SLEEP BOOSTER"   // DB27
{ S7_Optimized_Access := 'TRUE' }
AUTHOR : Simatic
FAMILY : IEC
NAME : IEC_TMR
VERSION : 1.0
// stored: InstanceOfName IEC_TIMER
"IEC_TIMER"
BEGIN
END_DATA_BLOCK

DATA_BLOCK "RESET SLEEP BOOSTER"   // DB28
{ S7_Optimized_Access := 'TRUE' }
AUTHOR : Simatic
FAMILY : IEC
NAME : IEC_TMR
VERSION : 1.0
// stored: InstanceOfName IEC_TIMER
"IEC_TIMER"
BEGIN
END_DATA_BLOCK

DATA_BLOCK "CONFIRMACION FLUJO 096P001A"   // DB31
{ S7_Optimized_Access := 'TRUE' }
AUTHOR : Simatic
FAMILY : IEC
NAME : IEC_TMR
VERSION : 1.0
// stored: InstanceOfName IEC_TIMER
"IEC_TIMER"
BEGIN
END_DATA_BLOCK

DATA_BLOCK "CONFIRMACION FLUJO 096P001B"   // DB32
{ S7_Optimized_Access := 'TRUE' }
AUTHOR : Simatic
FAMILY : IEC
NAME : IEC_TMR
VERSION : 1.0
// stored: InstanceOfName IEC_TIMER
"IEC_TIMER"
BEGIN
END_DATA_BLOCK

DATA_BLOCK "CONFIRMACION FLUJO 096P001C"   // DB33
{ S7_Optimized_Access := 'TRUE' }
AUTHOR : Simatic
FAMILY : IEC
NAME : IEC_TMR
VERSION : 1.0
// stored: InstanceOfName IEC_TIMER
"IEC_TIMER"
BEGIN
END_DATA_BLOCK

DATA_BLOCK "CONFIRMACION FLUJO 096P001D"   // DB34
{ S7_Optimized_Access := 'TRUE' }
AUTHOR : Simatic
FAMILY : IEC
NAME : IEC_TMR
VERSION : 1.0
// stored: InstanceOfName IEC_TIMER
"IEC_TIMER"
BEGIN
END_DATA_BLOCK

DATA_BLOCK "CONFIRMACION FLUJO 096P001E"   // DB35
{ S7_Optimized_Access := 'TRUE' }
AUTHOR : Simatic
FAMILY : IEC
NAME : IEC_TMR
VERSION : 1.0
// stored: InstanceOfName IEC_TIMER
"IEC_TIMER"
BEGIN
END_DATA_BLOCK

DATA_BLOCK "CONFIRMACION FLUJO 096P001F"   // DB36
{ S7_Optimized_Access := 'TRUE' }
AUTHOR : Simatic
FAMILY : IEC
NAME : IEC_TMR
VERSION : 1.0
// stored: InstanceOfName IEC_TIMER
"IEC_TIMER"
BEGIN
END_DATA_BLOCK

DATA_BLOCK "CONTADOR COMUNICACION"   // DB46
{ S7_Optimized_Access := 'TRUE' }
AUTHOR : Simatic
FAMILY : IEC
NAME : CNTR
VERSION : 1.0
// stored: InstanceOfName IEC_COUNTER
"IEC_COUNTER"
BEGIN
END_DATA_BLOCK

DATA_BLOCK "CONT SEG BA"   // DB53
{ S7_Optimized_Access := 'TRUE' }
AUTHOR : Simatic
FAMILY : IEC
NAME : CNTR
VERSION : 1.0
// stored: InstanceOfName IEC_COUNTER
"IEC_COUNTER"
BEGIN
END_DATA_BLOCK

DATA_BLOCK "CONT MIN BA"   // DB54
{ S7_Optimized_Access := 'TRUE' }
AUTHOR : Simatic
FAMILY : IEC
NAME : CNTR
VERSION : 1.0
// stored: InstanceOfName IEC_COUNTER
"IEC_COUNTER"
BEGIN
END_DATA_BLOCK

DATA_BLOCK "RESET BA"   // DB55
{ S7_Optimized_Access := 'TRUE' }
AUTHOR : Simatic
FAMILY : IEC
NAME : IEC_TMR
VERSION : 1.0
// stored: InstanceOfName IEC_TIMER
"IEC_TIMER"
BEGIN
END_DATA_BLOCK

DATA_BLOCK "CONT SEG BB"   // DB56
{ S7_Optimized_Access := 'TRUE' }
AUTHOR : Simatic
FAMILY : IEC
NAME : CNTR
VERSION : 1.0
// stored: InstanceOfName IEC_COUNTER
"IEC_COUNTER"
BEGIN
END_DATA_BLOCK

DATA_BLOCK "CONT MIN BB"   // DB57
{ S7_Optimized_Access := 'TRUE' }
AUTHOR : Simatic
FAMILY : IEC
NAME : CNTR
VERSION : 1.0
// stored: InstanceOfName IEC_COUNTER
"IEC_COUNTER"
BEGIN
END_DATA_BLOCK

DATA_BLOCK "RESET BB"   // DB58
{ S7_Optimized_Access := 'TRUE' }
AUTHOR : Simatic
FAMILY : IEC
NAME : IEC_TMR
VERSION : 1.0
// stored: InstanceOfName IEC_TIMER
"IEC_TIMER"
BEGIN
END_DATA_BLOCK

DATA_BLOCK "CONT SEG BC"   // DB59
{ S7_Optimized_Access := 'TRUE' }
AUTHOR : Simatic
FAMILY : IEC
NAME : CNTR
VERSION : 1.0
// stored: InstanceOfName IEC_COUNTER
"IEC_COUNTER"
BEGIN
END_DATA_BLOCK

DATA_BLOCK "CONT MIN BC"   // DB60
{ S7_Optimized_Access := 'TRUE' }
AUTHOR : Simatic
FAMILY : IEC
NAME : CNTR
VERSION : 1.0
// stored: InstanceOfName IEC_COUNTER
"IEC_COUNTER"
BEGIN
END_DATA_BLOCK

DATA_BLOCK "RESET BC"   // DB61
{ S7_Optimized_Access := 'TRUE' }
AUTHOR : Simatic
FAMILY : IEC
NAME : IEC_TMR
VERSION : 1.0
// stored: InstanceOfName IEC_TIMER
"IEC_TIMER"
BEGIN
END_DATA_BLOCK

DATA_BLOCK "CONT SEG BD"   // DB62
{ S7_Optimized_Access := 'TRUE' }
AUTHOR : Simatic
FAMILY : IEC
NAME : CNTR
VERSION : 1.0
// stored: InstanceOfName IEC_COUNTER
"IEC_COUNTER"
BEGIN
END_DATA_BLOCK

DATA_BLOCK "CONT MIN BD"   // DB63
{ S7_Optimized_Access := 'TRUE' }
AUTHOR : Simatic
FAMILY : IEC
NAME : CNTR
VERSION : 1.0
// stored: InstanceOfName IEC_COUNTER
"IEC_COUNTER"
BEGIN
END_DATA_BLOCK

DATA_BLOCK "RESET BD"   // DB64
{ S7_Optimized_Access := 'TRUE' }
AUTHOR : Simatic
FAMILY : IEC
NAME : IEC_TMR
VERSION : 1.0
// stored: InstanceOfName IEC_TIMER
"IEC_TIMER"
BEGIN
END_DATA_BLOCK

DATA_BLOCK "CONT SEG BE"   // DB65
{ S7_Optimized_Access := 'TRUE' }
AUTHOR : Simatic
FAMILY : IEC
NAME : CNTR
VERSION : 1.0
// stored: InstanceOfName IEC_COUNTER
"IEC_COUNTER"
BEGIN
END_DATA_BLOCK

DATA_BLOCK "CONT MIN BE"   // DB66
{ S7_Optimized_Access := 'TRUE' }
AUTHOR : Simatic
FAMILY : IEC
NAME : CNTR
VERSION : 1.0
// stored: InstanceOfName IEC_COUNTER
"IEC_COUNTER"
BEGIN
END_DATA_BLOCK

DATA_BLOCK "RESET BE"   // DB67
{ S7_Optimized_Access := 'TRUE' }
AUTHOR : Simatic
FAMILY : IEC
NAME : IEC_TMR
VERSION : 1.0
// stored: InstanceOfName IEC_TIMER
"IEC_TIMER"
BEGIN
END_DATA_BLOCK

DATA_BLOCK "CONT SEG BF"   // DB68
{ S7_Optimized_Access := 'TRUE' }
AUTHOR : Simatic
FAMILY : IEC
NAME : CNTR
VERSION : 1.0
// stored: InstanceOfName IEC_COUNTER
"IEC_COUNTER"
BEGIN
END_DATA_BLOCK

DATA_BLOCK "CONT MIN BF"   // DB69
{ S7_Optimized_Access := 'TRUE' }
AUTHOR : Simatic
FAMILY : IEC
NAME : CNTR
VERSION : 1.0
// stored: InstanceOfName IEC_COUNTER
"IEC_COUNTER"
BEGIN
END_DATA_BLOCK

DATA_BLOCK "RESET BF"   // DB70
{ S7_Optimized_Access := 'TRUE' }
AUTHOR : Simatic
FAMILY : IEC
NAME : IEC_TMR
VERSION : 1.0
// stored: InstanceOfName IEC_TIMER
"IEC_TIMER"
BEGIN
END_DATA_BLOCK

DATA_BLOCK "CONTADOR ALTERNACION"   // DB71
{ S7_Optimized_Access := 'TRUE' }
AUTHOR : Simatic
FAMILY : IEC
NAME : CNTR
VERSION : 1.0
// stored: InstanceOfName IEC_COUNTER
"IEC_COUNTER"
BEGIN
END_DATA_BLOCK

DATA_BLOCK "FALLA BOMBA LIDER 1"   // DB72
{ S7_Optimized_Access := 'TRUE' }
AUTHOR : Simatic
FAMILY : IEC
NAME : IEC_TMR
VERSION : 1.0
// stored: InstanceOfName IEC_TIMER
"IEC_TIMER"
BEGIN
END_DATA_BLOCK

DATA_BLOCK "FALLA BOMBA LIDER 6"   // DB73
{ S7_Optimized_Access := 'TRUE' }
AUTHOR : Simatic
FAMILY : IEC
NAME : IEC_TMR
VERSION : 1.0
// stored: InstanceOfName IEC_TIMER
"IEC_TIMER"
BEGIN
END_DATA_BLOCK

DATA_BLOCK "FALLA BOMBA LIDER 5"   // DB74
{ S7_Optimized_Access := 'TRUE' }
AUTHOR : Simatic
FAMILY : IEC
NAME : IEC_TMR
VERSION : 1.0
// stored: InstanceOfName IEC_TIMER
"IEC_TIMER"
BEGIN
END_DATA_BLOCK

DATA_BLOCK "FALLA BOMBA LIDER 4"   // DB75
{ S7_Optimized_Access := 'TRUE' }
AUTHOR : Simatic
FAMILY : IEC
NAME : IEC_TMR
VERSION : 1.0
// stored: InstanceOfName IEC_TIMER
"IEC_TIMER"
BEGIN
END_DATA_BLOCK

DATA_BLOCK "FALLA BOMBA LIDER 3"   // DB76
{ S7_Optimized_Access := 'TRUE' }
AUTHOR : Simatic
FAMILY : IEC
NAME : IEC_TMR
VERSION : 1.0
// stored: InstanceOfName IEC_TIMER
"IEC_TIMER"
BEGIN
END_DATA_BLOCK

DATA_BLOCK "FALLA BOMBA LIDER 2"   // DB77
{ S7_Optimized_Access := 'TRUE' }
AUTHOR : Simatic
FAMILY : IEC
NAME : IEC_TMR
VERSION : 1.0
// stored: InstanceOfName IEC_TIMER
"IEC_TIMER"
BEGIN
END_DATA_BLOCK

DATA_BLOCK "TIEMPO AD1"   // DB81
{ S7_Optimized_Access := 'TRUE' }
AUTHOR : Simatic
FAMILY : IEC
NAME : IEC_TMR
VERSION : 1.0
// stored: InstanceOfName IEC_TIMER
"IEC_TIMER"
BEGIN
END_DATA_BLOCK

DATA_BLOCK "TIEMPO AD2"   // DB82
{ S7_Optimized_Access := 'TRUE' }
AUTHOR : Simatic
FAMILY : IEC
NAME : IEC_TMR
VERSION : 1.0
// stored: InstanceOfName IEC_TIMER
"IEC_TIMER"
BEGIN
END_DATA_BLOCK

DATA_BLOCK "TIEMPO AD3"   // DB83
{ S7_Optimized_Access := 'TRUE' }
AUTHOR : Simatic
FAMILY : IEC
NAME : IEC_TMR
VERSION : 1.0
// stored: InstanceOfName IEC_TIMER
"IEC_TIMER"
BEGIN
END_DATA_BLOCK

DATA_BLOCK "TIEMPO AD4"   // DB84
{ S7_Optimized_Access := 'TRUE' }
AUTHOR : Simatic
FAMILY : IEC
NAME : IEC_TMR
VERSION : 1.0
// stored: InstanceOfName IEC_TIMER
"IEC_TIMER"
BEGIN
END_DATA_BLOCK

DATA_BLOCK "TIEMPO AD5"   // DB85
{ S7_Optimized_Access := 'TRUE' }
AUTHOR : Simatic
FAMILY : IEC
NAME : IEC_TMR
VERSION : 1.0
// stored: InstanceOfName IEC_TIMER
"IEC_TIMER"
BEGIN
END_DATA_BLOCK

DATA_BLOCK "PRES OK"   // DB86
{ S7_Optimized_Access := 'TRUE' }
AUTHOR : Simatic
FAMILY : IEC
NAME : IEC_TMR
VERSION : 1.0
// stored: InstanceOfName IEC_TIMER
"IEC_TIMER"
BEGIN
END_DATA_BLOCK

DATA_BLOCK "TOF1"   // DB87
{ S7_Optimized_Access := 'TRUE' }
AUTHOR : Simatic
FAMILY : IEC
NAME : IEC_TMR
VERSION : 1.0
// stored: InstanceOfName IEC_TIMER
"IEC_TIMER"
BEGIN
END_DATA_BLOCK

DATA_BLOCK "TOF2"   // DB88
{ S7_Optimized_Access := 'TRUE' }
AUTHOR : Simatic
FAMILY : IEC
NAME : IEC_TMR
VERSION : 1.0
// stored: InstanceOfName IEC_TIMER
"IEC_TIMER"
BEGIN
END_DATA_BLOCK

DATA_BLOCK "TOF3"   // DB89
{ S7_Optimized_Access := 'TRUE' }
AUTHOR : Simatic
FAMILY : IEC
NAME : IEC_TMR
VERSION : 1.0
// stored: InstanceOfName IEC_TIMER
"IEC_TIMER"
BEGIN
END_DATA_BLOCK

DATA_BLOCK "TOF4"   // DB90
{ S7_Optimized_Access := 'TRUE' }
AUTHOR : Simatic
FAMILY : IEC
NAME : IEC_TMR
VERSION : 1.0
// stored: InstanceOfName IEC_TIMER
"IEC_TIMER"
BEGIN
END_DATA_BLOCK

DATA_BLOCK "TOF5"   // DB91
{ S7_Optimized_Access := 'TRUE' }
AUTHOR : Simatic
FAMILY : IEC
NAME : IEC_TMR
VERSION : 1.0
// stored: InstanceOfName IEC_TIMER
"IEC_TIMER"
BEGIN
END_DATA_BLOCK

DATA_BLOCK "TOF6"   // DB92
{ S7_Optimized_Access := 'TRUE' }
AUTHOR : Simatic
FAMILY : IEC
NAME : IEC_TMR
VERSION : 1.0
// stored: InstanceOfName IEC_TIMER
"IEC_TIMER"
BEGIN
END_DATA_BLOCK

DATA_BLOCK "TIEMPO CONFIRMACION 096P001A"   // DB94
{ S7_Optimized_Access := 'TRUE' }
AUTHOR : Simatic
FAMILY : IEC
NAME : IEC_TMR
VERSION : 1.0
// stored: InstanceOfName IEC_TIMER
"IEC_TIMER"
BEGIN
END_DATA_BLOCK

DATA_BLOCK "TIEMPO CONFIRMACION 096P001B"   // DB95
{ S7_Optimized_Access := 'TRUE' }
AUTHOR : Simatic
FAMILY : IEC
NAME : IEC_TMR
VERSION : 1.0
// stored: InstanceOfName IEC_TIMER
"IEC_TIMER"
BEGIN
END_DATA_BLOCK

DATA_BLOCK "TIEMPO CONFIRMACION 096P001C"   // DB96
{ S7_Optimized_Access := 'TRUE' }
AUTHOR : Simatic
FAMILY : IEC
NAME : IEC_TMR
VERSION : 1.0
// stored: InstanceOfName IEC_TIMER
"IEC_TIMER"
BEGIN
END_DATA_BLOCK

DATA_BLOCK "TIEMPO CONFIRMACION 096P001D"   // DB97
{ S7_Optimized_Access := 'TRUE' }
AUTHOR : Simatic
FAMILY : IEC
NAME : IEC_TMR
VERSION : 1.0
// stored: InstanceOfName IEC_TIMER
"IEC_TIMER"
BEGIN
END_DATA_BLOCK

DATA_BLOCK "TIEMPO CONFIRMACION 096P001E"   // DB98
{ S7_Optimized_Access := 'TRUE' }
AUTHOR : Simatic
FAMILY : IEC
NAME : IEC_TMR
VERSION : 1.0
// stored: InstanceOfName IEC_TIMER
"IEC_TIMER"
BEGIN
END_DATA_BLOCK

DATA_BLOCK "TIEMPO CONFIRMACION 096P001F"   // DB99
{ S7_Optimized_Access := 'TRUE' }
AUTHOR : Simatic
FAMILY : IEC
NAME : IEC_TMR
VERSION : 1.0
// stored: InstanceOfName IEC_TIMER
"IEC_TIMER"
BEGIN
END_DATA_BLOCK

DATA_BLOCK "tiempo confirmacion presion"   // DB100
{ S7_Optimized_Access := 'TRUE' }
AUTHOR : Simatic
FAMILY : IEC
NAME : IEC_TMR
VERSION : 1.0
// stored: InstanceOfName IEC_TIMER
"IEC_TIMER"
BEGIN
END_DATA_BLOCK

DATA_BLOCK "CONT MIN BOMBA A ACUM"   // DB101
{ S7_Optimized_Access := 'TRUE' }
AUTHOR : Simatic
FAMILY : IEC
NAME : CNTR
VERSION : 1.0
// stored: InstanceOfName IEC_COUNTER
"IEC_COUNTER"
BEGIN
END_DATA_BLOCK

DATA_BLOCK "CONT H BOMBA A ACUM"   // DB102
{ S7_Optimized_Access := 'TRUE' }
AUTHOR : Simatic
FAMILY : IEC
NAME : CNTR
VERSION : 1.0
// stored: InstanceOfName IEC_COUNTER
"IEC_COUNTER"
BEGIN
END_DATA_BLOCK

DATA_BLOCK "CONT MIN BOMBA B ACUM"   // DB103
{ S7_Optimized_Access := 'TRUE' }
AUTHOR : Simatic
FAMILY : IEC
NAME : CNTR
VERSION : 1.0
// stored: InstanceOfName IEC_COUNTER
"IEC_COUNTER"
BEGIN
END_DATA_BLOCK

DATA_BLOCK "CONT H BOMBA B ACUM"   // DB104
{ S7_Optimized_Access := 'TRUE' }
AUTHOR : Simatic
FAMILY : IEC
NAME : CNTR
VERSION : 1.0
// stored: InstanceOfName IEC_COUNTER
"IEC_COUNTER"
BEGIN
END_DATA_BLOCK

DATA_BLOCK "CONT MIN BOMBA C ACUM"   // DB105
{ S7_Optimized_Access := 'TRUE' }
AUTHOR : Simatic
FAMILY : IEC
NAME : CNTR
VERSION : 1.0
// stored: InstanceOfName IEC_COUNTER
"IEC_COUNTER"
BEGIN
END_DATA_BLOCK

DATA_BLOCK "CONT H BOMBA C ACUM"   // DB106
{ S7_Optimized_Access := 'TRUE' }
AUTHOR : Simatic
FAMILY : IEC
NAME : CNTR
VERSION : 1.0
// stored: InstanceOfName IEC_COUNTER
"IEC_COUNTER"
BEGIN
END_DATA_BLOCK

DATA_BLOCK "CONT MIN BOMBA D ACUM"   // DB107
{ S7_Optimized_Access := 'TRUE' }
AUTHOR : Simatic
FAMILY : IEC
NAME : CNTR
VERSION : 1.0
// stored: InstanceOfName IEC_COUNTER
"IEC_COUNTER"
BEGIN
END_DATA_BLOCK

DATA_BLOCK "CONT H BOMBA D ACUM"   // DB108
{ S7_Optimized_Access := 'TRUE' }
AUTHOR : Simatic
FAMILY : IEC
NAME : CNTR
VERSION : 1.0
// stored: InstanceOfName IEC_COUNTER
"IEC_COUNTER"
BEGIN
END_DATA_BLOCK

DATA_BLOCK "CONT MIN BOMBA E ACUM"   // DB109
{ S7_Optimized_Access := 'TRUE' }
AUTHOR : Simatic
FAMILY : IEC
NAME : CNTR
VERSION : 1.0
// stored: InstanceOfName IEC_COUNTER
"IEC_COUNTER"
BEGIN
END_DATA_BLOCK

DATA_BLOCK "CONT H BOMBA E ACUM"   // DB110
{ S7_Optimized_Access := 'TRUE' }
AUTHOR : Simatic
FAMILY : IEC
NAME : CNTR
VERSION : 1.0
// stored: InstanceOfName IEC_COUNTER
"IEC_COUNTER"
BEGIN
END_DATA_BLOCK

DATA_BLOCK "CONT MIN BOMBA F ACUM"   // DB111
{ S7_Optimized_Access := 'TRUE' }
AUTHOR : Simatic
FAMILY : IEC
NAME : CNTR
VERSION : 1.0
// stored: InstanceOfName IEC_COUNTER
"IEC_COUNTER"
BEGIN
END_DATA_BLOCK

DATA_BLOCK "CONT H BOMBA F ACUM"   // DB112
{ S7_Optimized_Access := 'TRUE' }
AUTHOR : Simatic
FAMILY : IEC
NAME : CNTR
VERSION : 1.0
// stored: InstanceOfName IEC_COUNTER
"IEC_COUNTER"
BEGIN
END_DATA_BLOCK

DATA_BLOCK "RESET VFD1"   // DB113
{ S7_Optimized_Access := 'TRUE' }
AUTHOR : Simatic
FAMILY : IEC
NAME : IEC_TMR
VERSION : 1.0
// stored: InstanceOfName IEC_TIMER
"IEC_TIMER"
BEGIN
END_DATA_BLOCK

DATA_BLOCK "RESET VFD2"   // DB114
{ S7_Optimized_Access := 'TRUE' }
AUTHOR : Simatic
FAMILY : IEC
NAME : IEC_TMR
VERSION : 1.0
// stored: InstanceOfName IEC_TIMER
"IEC_TIMER"
BEGIN
END_DATA_BLOCK

DATA_BLOCK "RESET VFD3"   // DB115
{ S7_Optimized_Access := 'TRUE' }
AUTHOR : Simatic
FAMILY : IEC
NAME : IEC_TMR
VERSION : 1.0
// stored: InstanceOfName IEC_TIMER
"IEC_TIMER"
BEGIN
END_DATA_BLOCK

DATA_BLOCK "RESET VFD4"   // DB116
{ S7_Optimized_Access := 'TRUE' }
AUTHOR : Simatic
FAMILY : IEC
NAME : IEC_TMR
VERSION : 1.0
// stored: InstanceOfName IEC_TIMER
"IEC_TIMER"
BEGIN
END_DATA_BLOCK

DATA_BLOCK "RESET VFD5"   // DB117
{ S7_Optimized_Access := 'TRUE' }
AUTHOR : Simatic
FAMILY : IEC
NAME : IEC_TMR
VERSION : 1.0
// stored: InstanceOfName IEC_TIMER
"IEC_TIMER"
BEGIN
END_DATA_BLOCK

DATA_BLOCK "RESET VFD6"   // DB118
{ S7_Optimized_Access := 'TRUE' }
AUTHOR : Simatic
FAMILY : IEC
NAME : IEC_TMR
VERSION : 1.0
// stored: InstanceOfName IEC_TIMER
"IEC_TIMER"
BEGIN
END_DATA_BLOCK

// folder: (top level)

FUNCTION "Esc Entradas Analogas" : Void   // FC1, LAD
{ S7_Optimized_Access := 'TRUE' }
VERSION : 0.1
BEGIN

REGION Network 1: 096PIT001
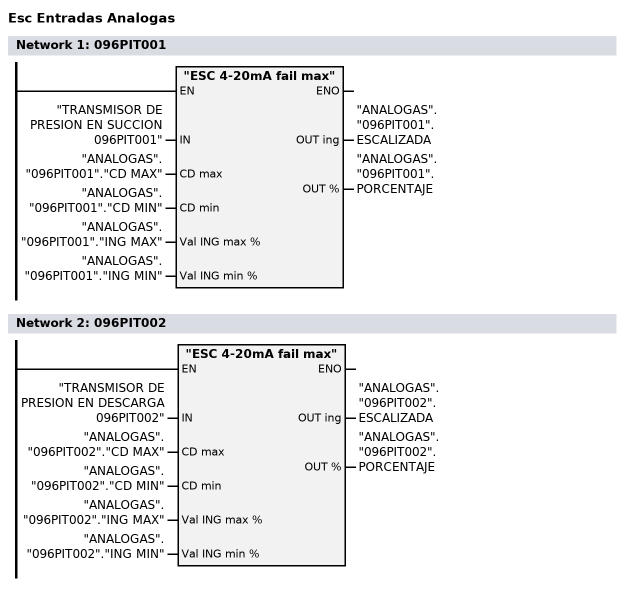
   RUNG wire#powerrail
      "ESC 4-20mA fail max"(IN := "TRANSMISOR DE PRESION EN SUCCION 096PIT001", "CD max" := "ANALOGAS"."096PIT001"."CD MAX", "CD min" := "ANALOGAS"."096PIT001"."CD MIN", "Val ING max %" := "ANALOGAS"."096PIT001"."ING MAX", "Val ING min %" := "ANALOGAS"."096PIT001"."ING MIN", "OUT ing" => "ANALOGAS"."096PIT001".ESCALIZADA, "OUT %" => "ANALOGAS"."096PIT001".PORCENTAJE)
   END_RUNG
   // the same network as SCL:
   "ESC 4-20mA fail max"(IN := "TRANSMISOR DE PRESION EN SUCCION 096PIT001",
                         "CD max" := "ANALOGAS"."096PIT001"."CD MAX",
                         "CD min" := "ANALOGAS"."096PIT001"."CD MIN",
                         "Val ING max %" := "ANALOGAS"."096PIT001"."ING MAX",
                         "Val ING min %" := "ANALOGAS"."096PIT001"."ING MIN",
                         "OUT ing" => "ANALOGAS"."096PIT001".ESCALIZADA,
                         "OUT %" => "ANALOGAS"."096PIT001".PORCENTAJE);
END_REGION

REGION Network 2: 096PIT002
   RUNG wire#powerrail
      "ESC 4-20mA fail max"(IN := "TRANSMISOR DE PRESION EN DESCARGA 096PIT002", "CD max" := "ANALOGAS"."096PIT002"."CD MAX", "CD min" := "ANALOGAS"."096PIT002"."CD MIN", "Val ING max %" := "ANALOGAS"."096PIT002"."ING MAX", "Val ING min %" := "ANALOGAS"."096PIT002"."ING MIN", "OUT ing" => "ANALOGAS"."096PIT002".ESCALIZADA, "OUT %" => "ANALOGAS"."096PIT002".PORCENTAJE)
   END_RUNG
   // the same network as SCL:
   "ESC 4-20mA fail max"(IN := "TRANSMISOR DE PRESION EN DESCARGA 096PIT002",
                         "CD max" := "ANALOGAS"."096PIT002"."CD MAX",
                         "CD min" := "ANALOGAS"."096PIT002"."CD MIN",
                         "Val ING max %" := "ANALOGAS"."096PIT002"."ING MAX",
                         "Val ING min %" := "ANALOGAS"."096PIT002"."ING MIN",
                         "OUT ing" => "ANALOGAS"."096PIT002".ESCALIZADA,
                         "OUT %" => "ANALOGAS"."096PIT002".PORCENTAJE);
END_REGION
END_FUNCTION

FUNCTION "ARRANQUE MOTORES" : Void   // FC2, LAD
{ S7_Optimized_Access := 'TRUE' }
VERSION : 0.1
   VAR_TEMP
      "SIN FLUJO SISTEMA 096P001A" : Bool;
      "SIN FLUJO SISTEMA 096P001B" : Bool;
      "SIN FLUJO SISTEMA 096P001C" : Bool;
      "SIN FLUJO SISTEMA 096P001D" : Bool;
      "SIN FLUJO SISTEMA 096P001E" : Bool;
      "SIN FLUJO SISTEMA 096P001F" : Bool;
   END_VAR
BEGIN

REGION Network 1
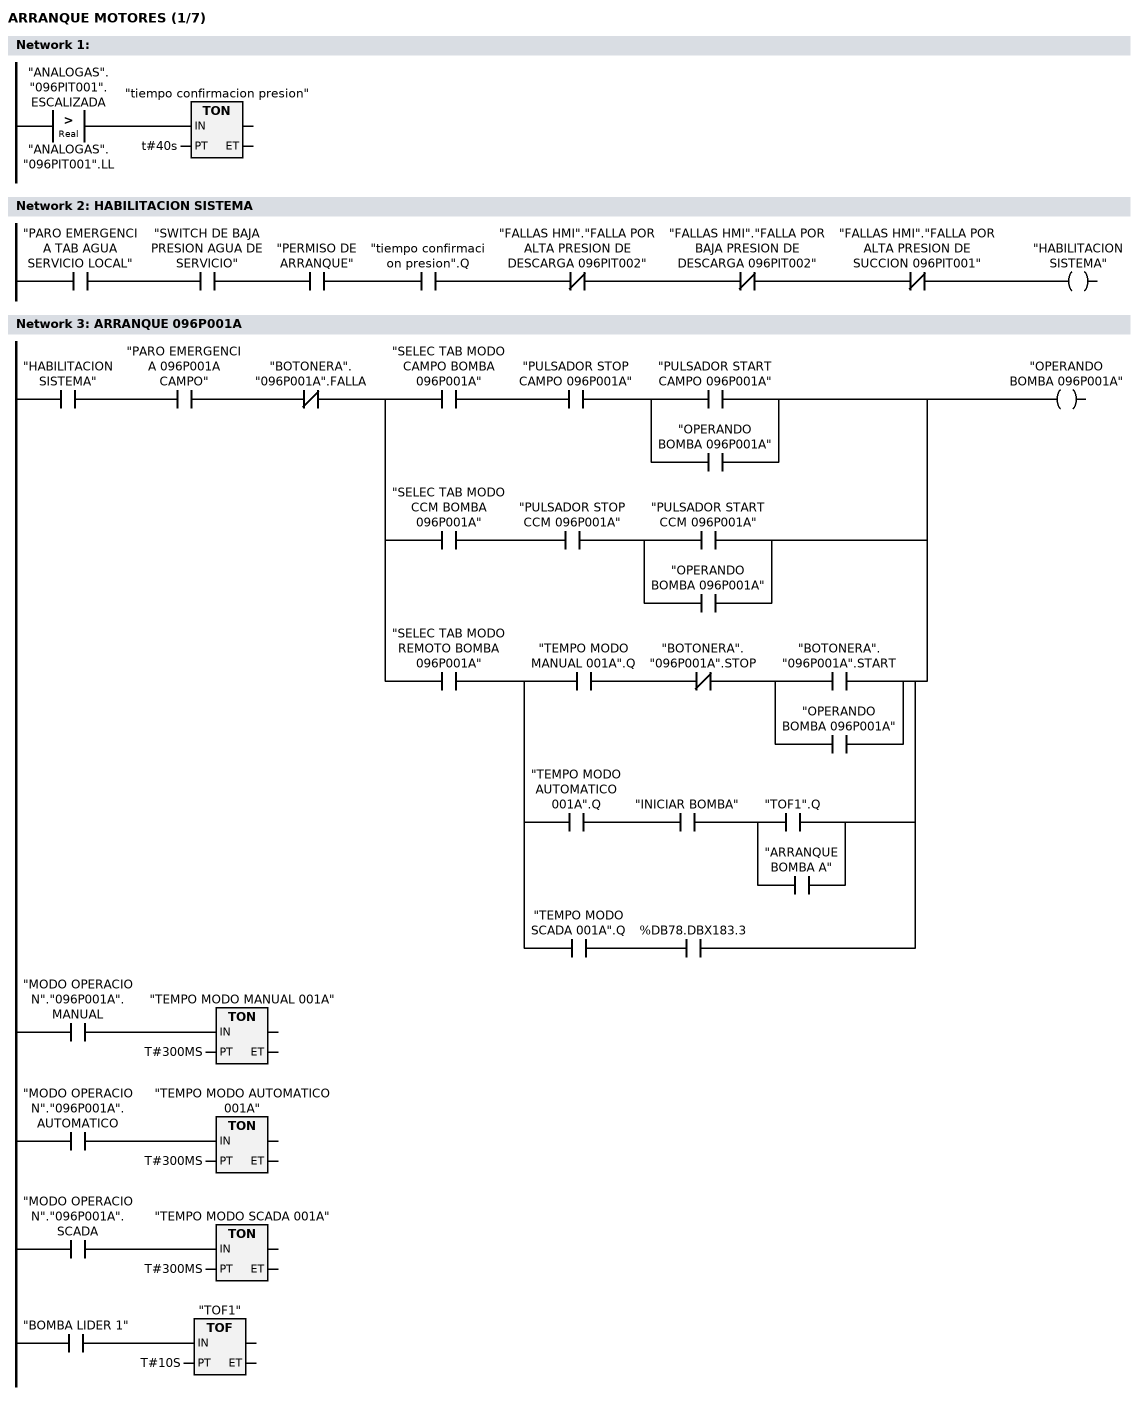
   "tiempo confirmacion presion".TON(IN := "ANALOGAS"."096PIT001".ESCALIZADA > "ANALOGAS"."096PIT001".LL,
                           PT := t#40s);
END_REGION

REGION Network 2: HABILITACION SISTEMA
   RUNG wire#powerrail
      Contact( "PARO EMERGENCIA TAB AGUA SERVICIO LOCAL" )
      Contact( "SWITCH DE BAJA PRESION AGUA DE SERVICIO" )
      Contact( "PERMISO DE ARRANQUE" )
      Contact( "tiempo confirmacion presion".Q )
      I_Contact( "FALLAS HMI"."FALLA POR ALTA PRESION DE DESCARGA 096PIT002" )
      I_Contact( "FALLAS HMI"."FALLA POR BAJA PRESION DE DESCARGA 096PIT002" )
      I_Contact( "FALLAS HMI"."FALLA POR ALTA PRESION DE SUCCION 096PIT001" )
      Coil( "HABILITACION SISTEMA" )
   END_RUNG
   // the same network as SCL:
   "HABILITACION SISTEMA" := "PARO EMERGENCIA TAB AGUA SERVICIO LOCAL" AND "SWITCH DE BAJA PRESION AGUA DE SERVICIO" AND "PERMISO DE ARRANQUE" AND "tiempo confirmacion presion".Q AND NOT "FALLAS HMI"."FALLA POR ALTA PRESION DE DESCARGA 096PIT002" AND NOT "FALLAS HMI"."FALLA POR BAJA PRESION DE DESCARGA 096PIT002" AND NOT "FALLAS HMI"."FALLA POR ALTA PRESION DE SUCCION 096PIT001";
END_REGION

REGION Network 3: ARRANQUE 096P001A
   "OPERANDO BOMBA 096P001A" := "HABILITACION SISTEMA" AND "PARO EMERGENCIA 096P001A CAMPO" AND NOT "BOTONERA"."096P001A".FALLA AND (("SELEC TAB MODO CAMPO BOMBA 096P001A" AND "PULSADOR STOP CAMPO 096P001A" AND ("PULSADOR START CAMPO 096P001A" OR "OPERANDO BOMBA 096P001A")) OR ("SELEC TAB MODO CCM BOMBA 096P001A" AND "PULSADOR STOP CCM 096P001A" AND ("PULSADOR START CCM 096P001A" OR "OPERANDO BOMBA 096P001A")) OR ("SELEC TAB MODO REMOTO BOMBA 096P001A" AND (("TEMPO MODO MANUAL 001A".Q AND NOT "BOTONERA"."096P001A".STOP AND ("BOTONERA"."096P001A".START OR "OPERANDO BOMBA 096P001A")) OR ("TEMPO MODO AUTOMATICO 001A".Q AND "INICIAR BOMBA" AND ("TOF1".Q OR "ARRANQUE BOMBA A")) OR ("TEMPO MODO SCADA 001A".Q AND %DB78.DBX183.3))));
   "TEMPO MODO MANUAL 001A".TON(IN := "MODO OPERACION"."096P001A".MANUAL, PT := T#300MS);
   "TEMPO MODO AUTOMATICO 001A".TON(IN := "MODO OPERACION"."096P001A".AUTOMATICO, PT := T#300MS);
   "TEMPO MODO SCADA 001A".TON(IN := "MODO OPERACION"."096P001A".SCADA, PT := T#300MS);
   "TOF1".TOF(IN := "BOMBA LIDER 1", PT := T#10S);
END_REGION

REGION Network 4: ARRANQUE 096P001B
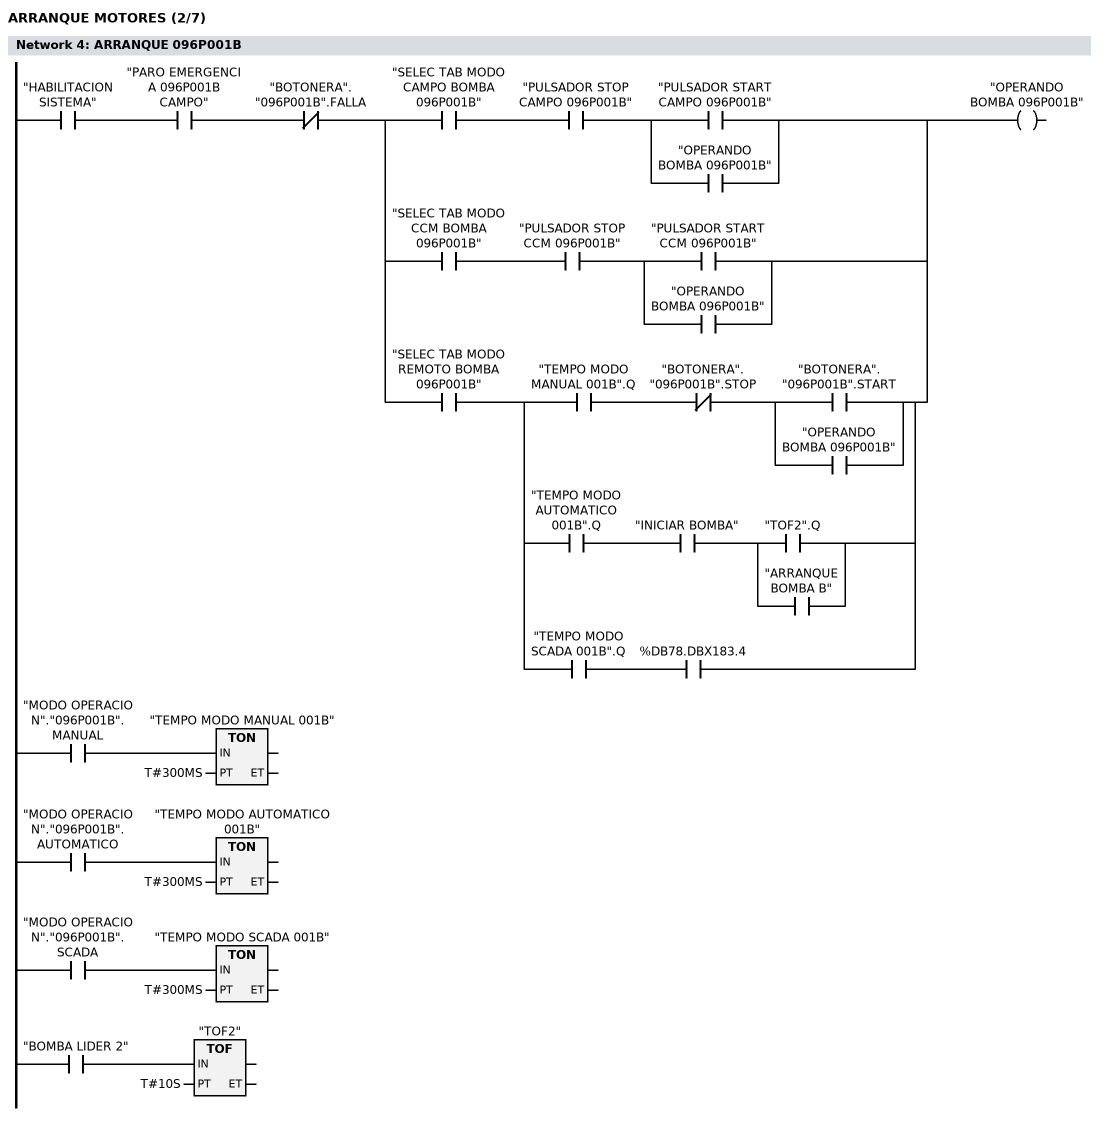
   "OPERANDO BOMBA 096P001B" := "HABILITACION SISTEMA" AND "PARO EMERGENCIA 096P001B CAMPO" AND NOT "BOTONERA"."096P001B".FALLA AND (("SELEC TAB MODO CAMPO BOMBA 096P001B" AND "PULSADOR STOP CAMPO 096P001B" AND ("PULSADOR START CAMPO 096P001B" OR "OPERANDO BOMBA 096P001B")) OR ("SELEC TAB MODO CCM BOMBA 096P001B" AND "PULSADOR STOP CCM 096P001B" AND ("PULSADOR START CCM 096P001B" OR "OPERANDO BOMBA 096P001B")) OR ("SELEC TAB MODO REMOTO BOMBA 096P001B" AND (("TEMPO MODO MANUAL 001B".Q AND NOT "BOTONERA"."096P001B".STOP AND ("BOTONERA"."096P001B".START OR "OPERANDO BOMBA 096P001B")) OR ("TEMPO MODO AUTOMATICO 001B".Q AND "INICIAR BOMBA" AND ("TOF2".Q OR "ARRANQUE BOMBA B")) OR ("TEMPO MODO SCADA 001B".Q AND %DB78.DBX183.4))));
   "TEMPO MODO MANUAL 001B".TON(IN := "MODO OPERACION"."096P001B".MANUAL, PT := T#300MS);
   "TEMPO MODO AUTOMATICO 001B".TON(IN := "MODO OPERACION"."096P001B".AUTOMATICO, PT := T#300MS);
   "TEMPO MODO SCADA 001B".TON(IN := "MODO OPERACION"."096P001B".SCADA, PT := T#300MS);
   "TOF2".TOF(IN := "BOMBA LIDER 2", PT := T#10S);
END_REGION

REGION Network 5: ARRANQUE 096P001C
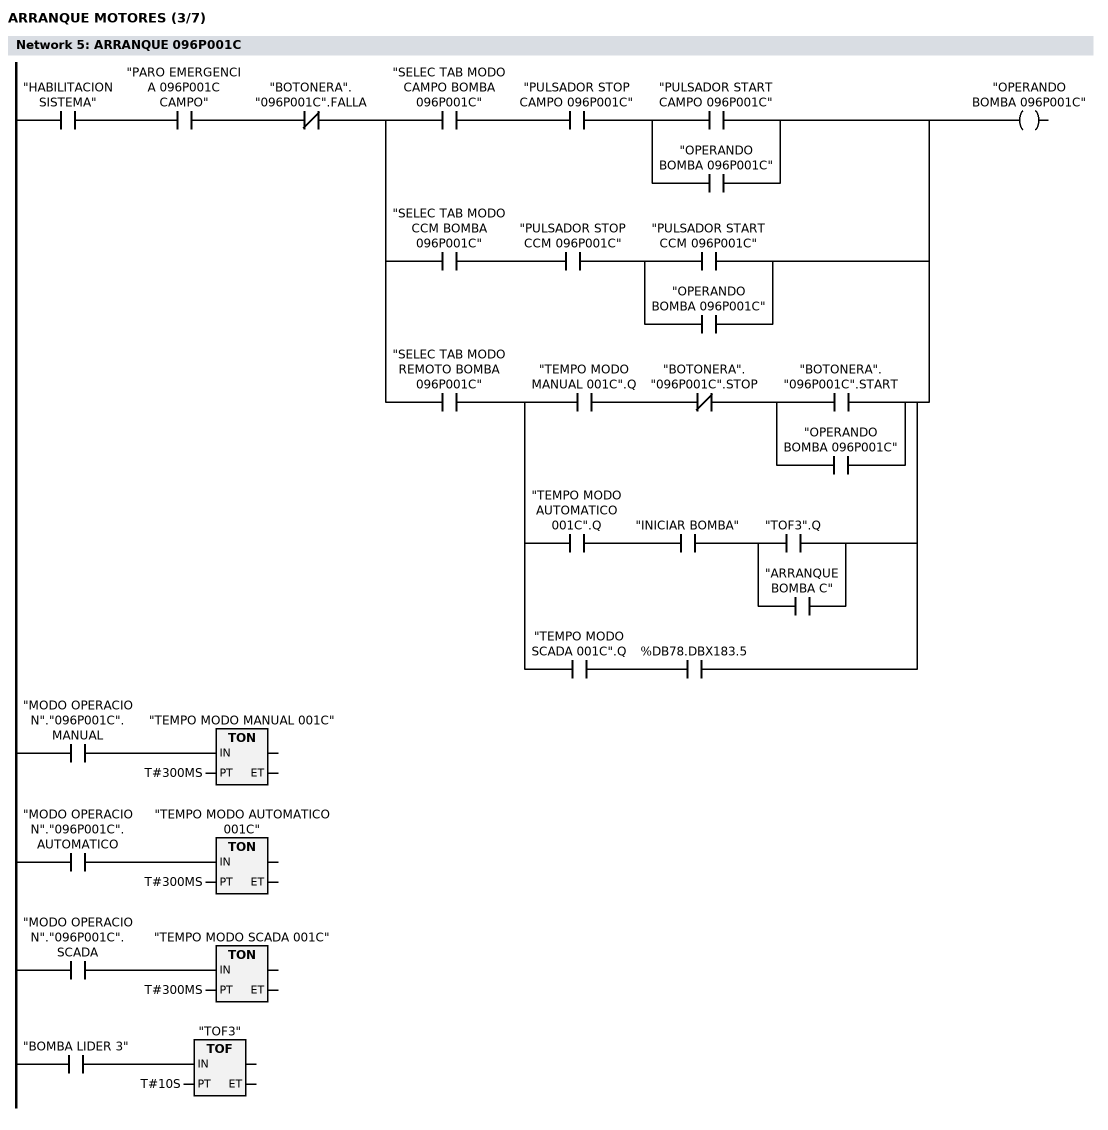
   "OPERANDO BOMBA 096P001C" := "HABILITACION SISTEMA" AND "PARO EMERGENCIA 096P001C CAMPO" AND NOT "BOTONERA"."096P001C".FALLA AND (("SELEC TAB MODO CAMPO BOMBA 096P001C" AND "PULSADOR STOP CAMPO 096P001C" AND ("PULSADOR START CAMPO 096P001C" OR "OPERANDO BOMBA 096P001C")) OR ("SELEC TAB MODO CCM BOMBA 096P001C" AND "PULSADOR STOP CCM 096P001C" AND ("PULSADOR START CCM 096P001C" OR "OPERANDO BOMBA 096P001C")) OR ("SELEC TAB MODO REMOTO BOMBA 096P001C" AND (("TEMPO MODO MANUAL 001C".Q AND NOT "BOTONERA"."096P001C".STOP AND ("BOTONERA"."096P001C".START OR "OPERANDO BOMBA 096P001C")) OR ("TEMPO MODO AUTOMATICO 001C".Q AND "INICIAR BOMBA" AND ("TOF3".Q OR "ARRANQUE BOMBA C")) OR ("TEMPO MODO SCADA 001C".Q AND %DB78.DBX183.5))));
   "TEMPO MODO MANUAL 001C".TON(IN := "MODO OPERACION"."096P001C".MANUAL, PT := T#300MS);
   "TEMPO MODO AUTOMATICO 001C".TON(IN := "MODO OPERACION"."096P001C".AUTOMATICO, PT := T#300MS);
   "TEMPO MODO SCADA 001C".TON(IN := "MODO OPERACION"."096P001C".SCADA, PT := T#300MS);
   "TOF3".TOF(IN := "BOMBA LIDER 3", PT := T#10S);
END_REGION

REGION Network 6: ARRANQUE 096P001D
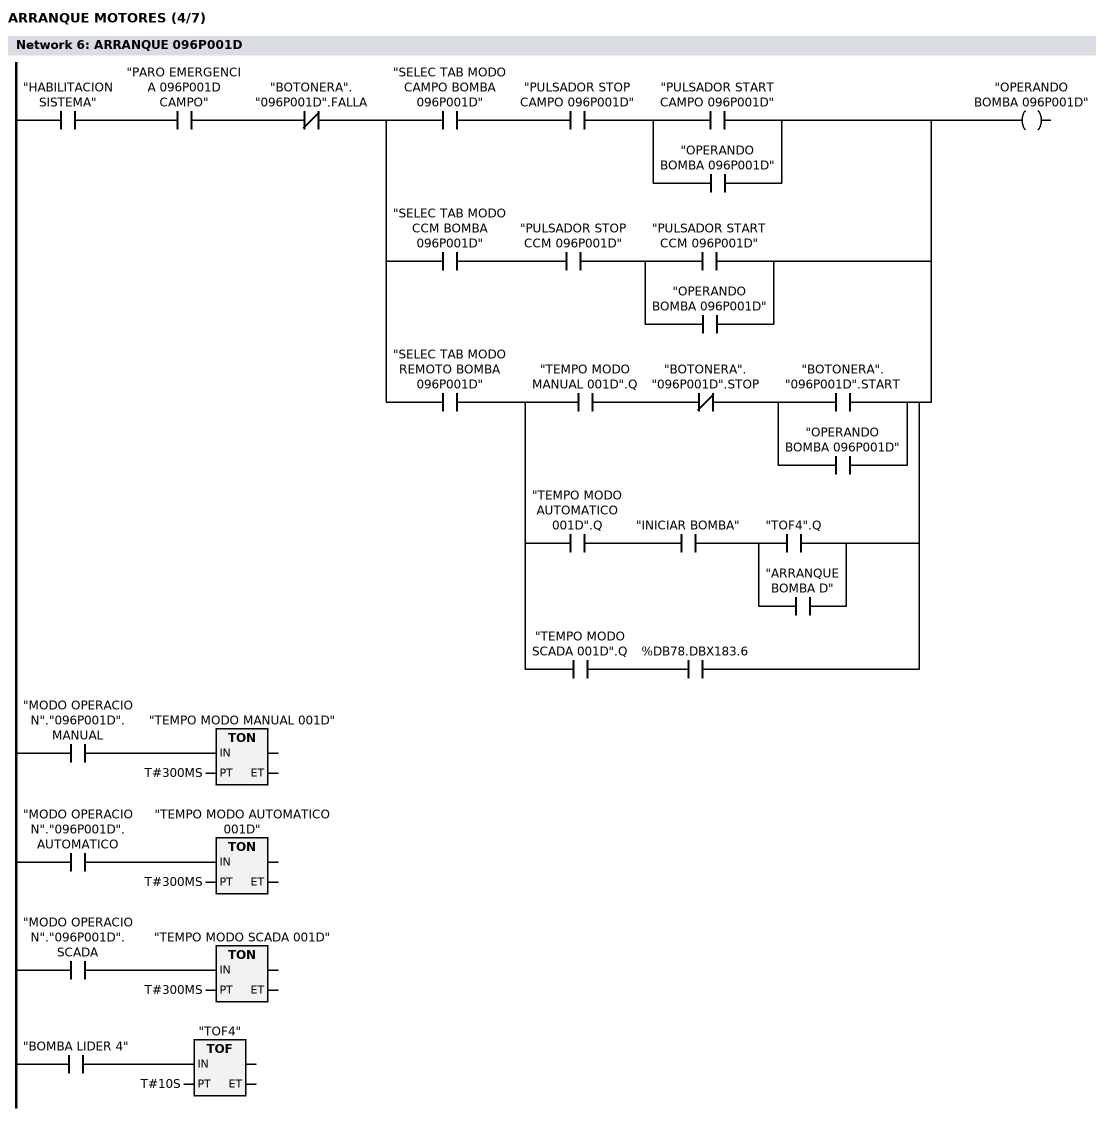
   "OPERANDO BOMBA 096P001D" := "HABILITACION SISTEMA" AND "PARO EMERGENCIA 096P001D CAMPO" AND NOT "BOTONERA"."096P001D".FALLA AND (("SELEC TAB MODO CAMPO BOMBA 096P001D" AND "PULSADOR STOP CAMPO 096P001D" AND ("PULSADOR START CAMPO 096P001D" OR "OPERANDO BOMBA 096P001D")) OR ("SELEC TAB MODO CCM BOMBA 096P001D" AND "PULSADOR STOP CCM 096P001D" AND ("PULSADOR START CCM 096P001D" OR "OPERANDO BOMBA 096P001D")) OR ("SELEC TAB MODO REMOTO BOMBA 096P001D" AND (("TEMPO MODO MANUAL 001D".Q AND NOT "BOTONERA"."096P001D".STOP AND ("BOTONERA"."096P001D".START OR "OPERANDO BOMBA 096P001D")) OR ("TEMPO MODO AUTOMATICO 001D".Q AND "INICIAR BOMBA" AND ("TOF4".Q OR "ARRANQUE BOMBA D")) OR ("TEMPO MODO SCADA 001D".Q AND %DB78.DBX183.6))));
   "TEMPO MODO MANUAL 001D".TON(IN := "MODO OPERACION"."096P001D".MANUAL, PT := T#300MS);
   "TEMPO MODO AUTOMATICO 001D".TON(IN := "MODO OPERACION"."096P001D".AUTOMATICO, PT := T#300MS);
   "TEMPO MODO SCADA 001D".TON(IN := "MODO OPERACION"."096P001D".SCADA, PT := T#300MS);
   "TOF4".TOF(IN := "BOMBA LIDER 4", PT := T#10S);
END_REGION

REGION Network 7: ARRANQUE 096P001E
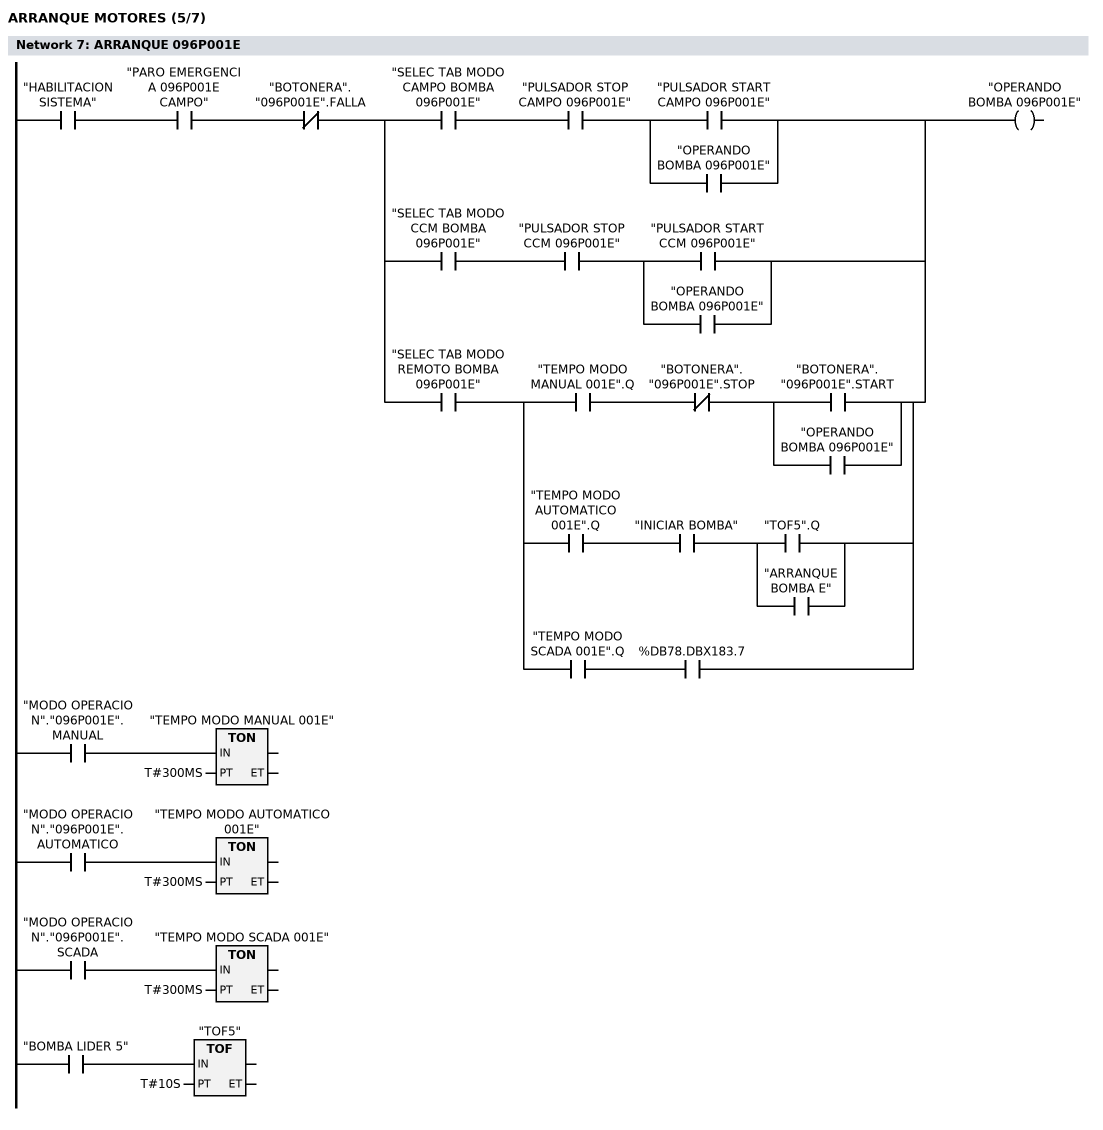
   "OPERANDO BOMBA 096P001E" := "HABILITACION SISTEMA" AND "PARO EMERGENCIA 096P001E CAMPO" AND NOT "BOTONERA"."096P001E".FALLA AND (("SELEC TAB MODO CAMPO BOMBA 096P001E" AND "PULSADOR STOP CAMPO 096P001E" AND ("PULSADOR START CAMPO 096P001E" OR "OPERANDO BOMBA 096P001E")) OR ("SELEC TAB MODO CCM BOMBA 096P001E" AND "PULSADOR STOP CCM 096P001E" AND ("PULSADOR START CCM 096P001E" OR "OPERANDO BOMBA 096P001E")) OR ("SELEC TAB MODO REMOTO BOMBA 096P001E" AND (("TEMPO MODO MANUAL 001E".Q AND NOT "BOTONERA"."096P001E".STOP AND ("BOTONERA"."096P001E".START OR "OPERANDO BOMBA 096P001E")) OR ("TEMPO MODO AUTOMATICO 001E".Q AND "INICIAR BOMBA" AND ("TOF5".Q OR "ARRANQUE BOMBA E")) OR ("TEMPO MODO SCADA 001E".Q AND %DB78.DBX183.7))));
   "TEMPO MODO MANUAL 001E".TON(IN := "MODO OPERACION"."096P001E".MANUAL, PT := T#300MS);
   "TEMPO MODO AUTOMATICO 001E".TON(IN := "MODO OPERACION"."096P001E".AUTOMATICO, PT := T#300MS);
   "TEMPO MODO SCADA 001E".TON(IN := "MODO OPERACION"."096P001E".SCADA, PT := T#300MS);
   "TOF5".TOF(IN := "BOMBA LIDER 5", PT := T#10S);
END_REGION

REGION Network 8: ARRANQUE 096P001F
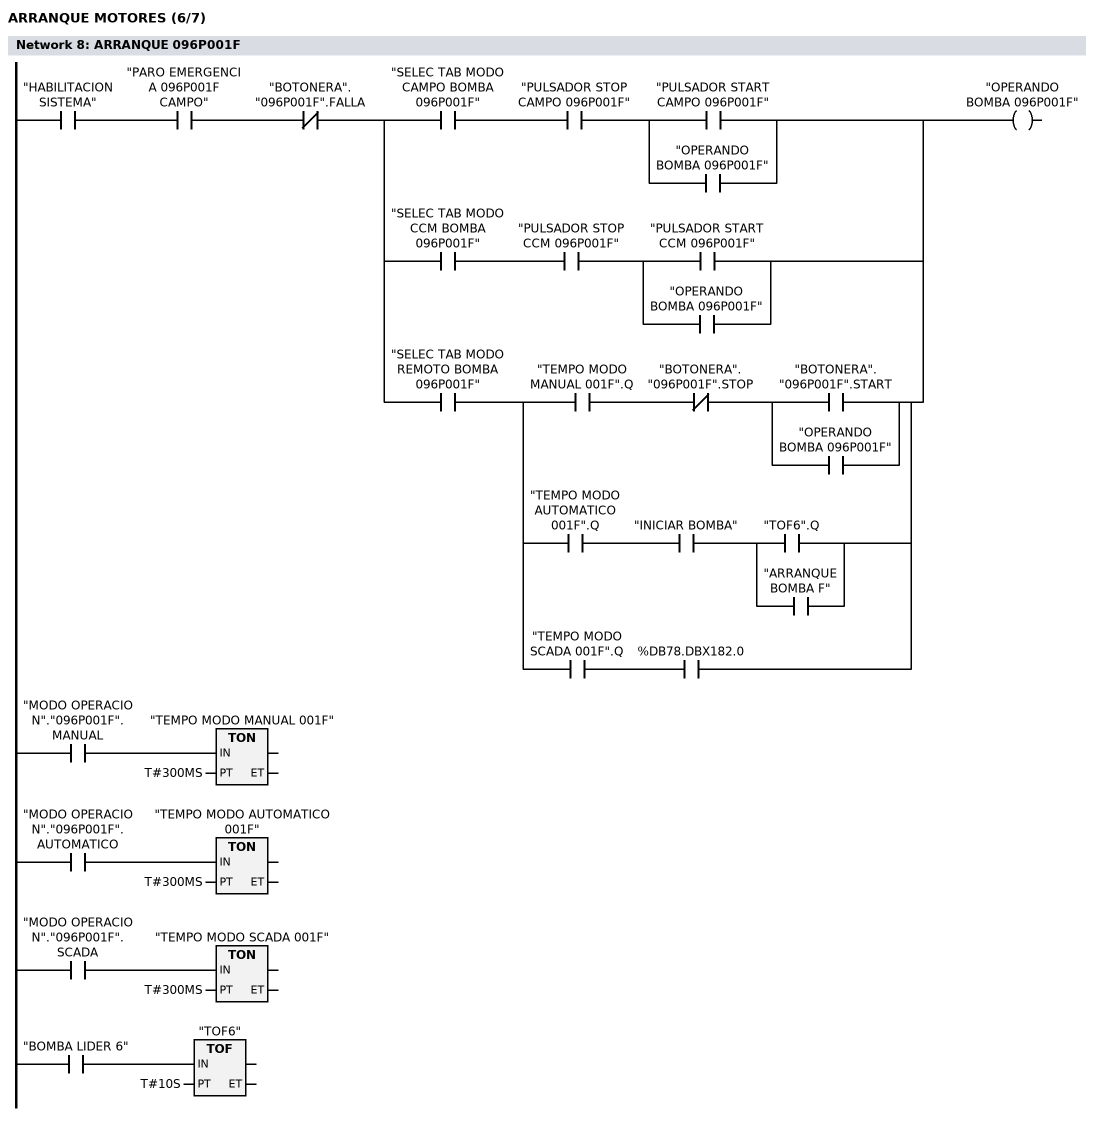
   "OPERANDO BOMBA 096P001F" := "HABILITACION SISTEMA" AND "PARO EMERGENCIA 096P001F CAMPO" AND NOT "BOTONERA"."096P001F".FALLA AND (("SELEC TAB MODO CAMPO BOMBA 096P001F" AND "PULSADOR STOP CAMPO 096P001F" AND ("PULSADOR START CAMPO 096P001F" OR "OPERANDO BOMBA 096P001F")) OR ("SELEC TAB MODO CCM BOMBA 096P001F" AND "PULSADOR STOP CCM 096P001F" AND ("PULSADOR START CCM 096P001F" OR "OPERANDO BOMBA 096P001F")) OR ("SELEC TAB MODO REMOTO BOMBA 096P001F" AND (("TEMPO MODO MANUAL 001F".Q AND NOT "BOTONERA"."096P001F".STOP AND ("BOTONERA"."096P001F".START OR "OPERANDO BOMBA 096P001F")) OR ("TEMPO MODO AUTOMATICO 001F".Q AND "INICIAR BOMBA" AND ("TOF6".Q OR "ARRANQUE BOMBA F")) OR ("TEMPO MODO SCADA 001F".Q AND %DB78.DBX182.0))));
   "TEMPO MODO MANUAL 001F".TON(IN := "MODO OPERACION"."096P001F".MANUAL, PT := T#300MS);
   "TEMPO MODO AUTOMATICO 001F".TON(IN := "MODO OPERACION"."096P001F".AUTOMATICO, PT := T#300MS);
   "TEMPO MODO SCADA 001F".TON(IN := "MODO OPERACION"."096P001F".SCADA, PT := T#300MS);
   "TOF6".TOF(IN := "BOMBA LIDER 6", PT := T#10S);
END_REGION

REGION Network 9: DISPONIBILIDAD DE BOMBAS
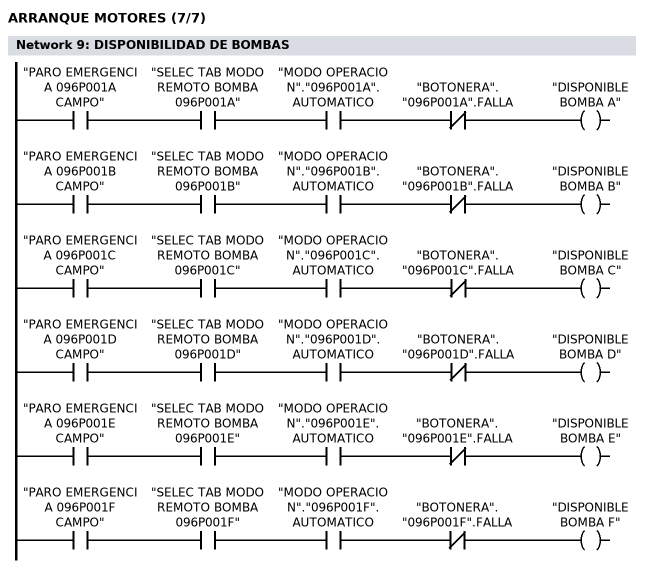
   RUNG wire#powerrail
      Contact( "PARO EMERGENCIA 096P001A CAMPO" )
      Contact( "SELEC TAB MODO REMOTO BOMBA 096P001A" )
      Contact( "MODO OPERACION"."096P001A".AUTOMATICO )
      I_Contact( "BOTONERA"."096P001A".FALLA )
      Coil( "DISPONIBLE BOMBA A" )
   END_RUNG
   RUNG wire#powerrail
      Contact( "PARO EMERGENCIA 096P001B CAMPO" )
      Contact( "SELEC TAB MODO REMOTO BOMBA 096P001B" )
      Contact( "MODO OPERACION"."096P001B".AUTOMATICO )
      I_Contact( "BOTONERA"."096P001B".FALLA )
      Coil( "DISPONIBLE BOMBA B" )
   END_RUNG
   RUNG wire#powerrail
      Contact( "PARO EMERGENCIA 096P001C CAMPO" )
      Contact( "SELEC TAB MODO REMOTO BOMBA 096P001C" )
      Contact( "MODO OPERACION"."096P001C".AUTOMATICO )
      I_Contact( "BOTONERA"."096P001C".FALLA )
      Coil( "DISPONIBLE BOMBA C" )
   END_RUNG
   RUNG wire#powerrail
      Contact( "PARO EMERGENCIA 096P001D CAMPO" )
      Contact( "SELEC TAB MODO REMOTO BOMBA 096P001D" )
      Contact( "MODO OPERACION"."096P001D".AUTOMATICO )
      I_Contact( "BOTONERA"."096P001D".FALLA )
      Coil( "DISPONIBLE BOMBA D" )
   END_RUNG
   RUNG wire#powerrail
      Contact( "PARO EMERGENCIA 096P001E CAMPO" )
      Contact( "SELEC TAB MODO REMOTO BOMBA 096P001E" )
      Contact( "MODO OPERACION"."096P001E".AUTOMATICO )
      I_Contact( "BOTONERA"."096P001E".FALLA )
      Coil( "DISPONIBLE BOMBA E" )
   END_RUNG
   RUNG wire#powerrail
      Contact( "PARO EMERGENCIA 096P001F CAMPO" )
      Contact( "SELEC TAB MODO REMOTO BOMBA 096P001F" )
      Contact( "MODO OPERACION"."096P001F".AUTOMATICO )
      I_Contact( "BOTONERA"."096P001F".FALLA )
      Coil( "DISPONIBLE BOMBA F" )
   END_RUNG
   // the same network as SCL:
   "DISPONIBLE BOMBA A" := "PARO EMERGENCIA 096P001A CAMPO" AND "SELEC TAB MODO REMOTO BOMBA 096P001A" AND "MODO OPERACION"."096P001A".AUTOMATICO AND NOT "BOTONERA"."096P001A".FALLA;
   "DISPONIBLE BOMBA B" := "PARO EMERGENCIA 096P001B CAMPO" AND "SELEC TAB MODO REMOTO BOMBA 096P001B" AND "MODO OPERACION"."096P001B".AUTOMATICO AND NOT "BOTONERA"."096P001B".FALLA;
   "DISPONIBLE BOMBA C" := "PARO EMERGENCIA 096P001C CAMPO" AND "SELEC TAB MODO REMOTO BOMBA 096P001C" AND "MODO OPERACION"."096P001C".AUTOMATICO AND NOT "BOTONERA"."096P001C".FALLA;
   "DISPONIBLE BOMBA D" := "PARO EMERGENCIA 096P001D CAMPO" AND "SELEC TAB MODO REMOTO BOMBA 096P001D" AND "MODO OPERACION"."096P001D".AUTOMATICO AND NOT "BOTONERA"."096P001D".FALLA;
   "DISPONIBLE BOMBA E" := "PARO EMERGENCIA 096P001E CAMPO" AND "SELEC TAB MODO REMOTO BOMBA 096P001E" AND "MODO OPERACION"."096P001E".AUTOMATICO AND NOT "BOTONERA"."096P001E".FALLA;
   "DISPONIBLE BOMBA F" := "PARO EMERGENCIA 096P001F CAMPO" AND "SELEC TAB MODO REMOTO BOMBA 096P001F" AND "MODO OPERACION"."096P001F".AUTOMATICO AND NOT "BOTONERA"."096P001F".FALLA;
END_REGION
END_FUNCTION

FUNCTION "ESC 4-20mA fail max" : Void   // FC3, LAD
{ S7_Optimized_Access := 'TRUE' }
VERSION : 0.1
   VAR_INPUT
      IN : Word;
      "CD max" : Real;
      "CD min" : Real;
      "Val ING max %" : Real;
      "Val ING min %" : Real;
   END_VAR
   VAR_OUTPUT
      "OUT ing" : Real;
      "OUT %" : Real;
   END_VAR
   VAR_TEMP
      "IN Real" : Real;
      "IN ok" : Real;
      "IN error <" : Bool;
      "IN error >" : Bool;
      "IN ESC" : Real;
      Temp_1 : Int;
   END_VAR
BEGIN

REGION Network 1
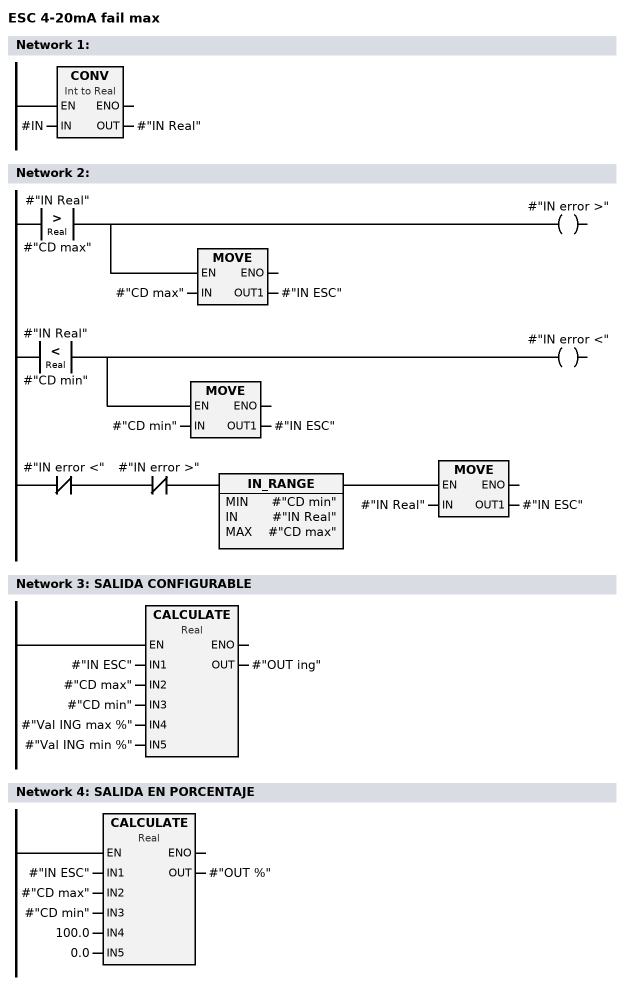
   RUNG wire#powerrail
      { S7_Templates := "[SrcType := Int, DestType := Real]" } Convert(in := #IN, out => #"IN Real")
   END_RUNG
   // the same network as SCL:
   #"IN Real" := INT_TO_REAL(#IN);
END_REGION

REGION Network 2
   RUNG wire#powerrail
      { S7_Templates := "SrcType := Real" } GT_Contact(in1 := #"IN Real", in2 := #"CD max")
      wire#w1
      Coil( #"IN error >" )
   END_RUNG
   RUNG wire#w1
      Move(in := #"CD max", out1 => #"IN ESC")
   END_RUNG
   RUNG wire#powerrail
      { S7_Templates := "SrcType := Real" } LT_Contact(in1 := #"IN Real", in2 := #"CD min")
      wire#w2
      Coil( #"IN error <" )
   END_RUNG
   RUNG wire#w2
      Move(in := #"CD min", out1 => #"IN ESC")
   END_RUNG
   RUNG wire#powerrail
      I_Contact( #"IN error <" )
      I_Contact( #"IN error >" )
      { S7_Templates := "SrcType := Real" } InRange(min := #"CD min", in := #"IN Real", max := #"CD max")
      Move(in := #"IN Real", out1 => #"IN ESC")
   END_RUNG
   // the same network as SCL:
   #"IN error >" := #"IN Real" > #"CD max";
   IF #"IN error >" THEN #"IN ESC" := #"CD max"; END_IF;
   #"IN error <" := #"IN Real" < #"CD min";
   IF #"IN error <" THEN #"IN ESC" := #"CD min"; END_IF;
   IF NOT #"IN error <" AND NOT #"IN error >" AND (#"CD min" <= #"IN Real") AND (#"IN Real" <= #"CD max") THEN
       #"IN ESC" := #"IN Real";
   END_IF;
END_REGION

REGION Network 3: SALIDA CONFIGURABLE
   RUNG wire#powerrail
      { S7_Templates := "SrcType := Real"; S7_Expression := "(((in4-in5)/(in2-in3))*in1)+(in5-(((in4-in5)/(in2-in3))*in3))" } Calculate(in1 := #"IN ESC", in2 := #"CD max", in3 := #"CD min", in4 := #"Val ING max %", in5 := #"Val ING min %", out => #"OUT ing")
   END_RUNG
   // the same network as SCL:
   #"OUT ing" := (((#"Val ING max %"-#"Val ING min %")/(#"CD max"-#"CD min"))*#"IN ESC")+(#"Val ING min %"-(((#"Val ING max %"-#"Val ING min %")/(#"CD max"-#"CD min"))*#"CD min"));
END_REGION

REGION Network 4: SALIDA EN PORCENTAJE
   RUNG wire#powerrail
      { S7_Templates := "SrcType := Real"; S7_Expression := "(((in4-in5)/(in2-in3))*in1)+(in5-(((in4-in5)/(in2-in3))*in3))" } Calculate(in1 := #"IN ESC", in2 := #"CD max", in3 := #"CD min", in4 := 100.0, in5 := 0.0, out => #"OUT %")
   END_RUNG
   // the same network as SCL:
   #"OUT %" := (((100.0-0.0)/(#"CD max"-#"CD min"))*#"IN ESC")+(0.0-(((100.0-0.0)/(#"CD max"-#"CD min"))*#"CD min"));
END_REGION

REGION Network 5: SALIDA EN mA
END_REGION
END_FUNCTION

FUNCTION "SISTEMA DE PRESION" : Void   // FC4, LAD
{ S7_Optimized_Access := 'TRUE' }
VERSION : 0.1
   VAR_TEMP
      T1 : Real;
      T2 : Real;
      T3 : Real;
      T4 : Real;
      T5 : Real;
      T6 : Real;
      t7 : Real;
      "Tiempo 1" : DInt;
      "Tiempo 2" : DInt;
      "Tiempo 3" : DInt;
      "Tiempo 4" : DInt;
      "Tiempo 5" : DInt;
      "Tiempo 6" : DInt;
      "Tiempo 7" : DInt;
      "DIFERENCIAL ARRANQUE" : Real;
      "DIFERENCIAL DORMIR" : Real;
      "FRECUENCIA OPERACION" : Real;
      ADICION : Bool;
      ACTIVAR : Bool;
      "SIN BOMBAS" : Bool;
      "Tiempo cumplido B1" : Bool;
      "Tiempo cumplido B2" : Bool;
      "Tiempo cumplido B3" : Bool;
      "Tiempo cumplido B4" : Bool;
      "Tiempo cumplido B5" : Bool;
      "Tiempo cumplido B6" : Bool;
      TEST1 : Bool;
      TEST2 : Bool;
      TEST3 : Bool;
      TEST4 : Bool;
      TEST5 : Bool;
      TEST6 : Bool;
      TEST7 : Bool;
      TEST8 : Bool;
      TEST9 : Bool;
      TEST10 : Bool;
      TEST11 : Bool;
      TEST12 : Bool;
   END_VAR
   VAR_TEMP   // added for the SCL form of the ladder/FBD networks
      _w1 : Bool;
      _w2 : Bool;
      _w3 : Bool;
      _w4 : Bool;
      _w5 : Bool;
      _w6 : Bool;
      _w7 : Bool;
      _w8 : Bool;
      _w9 : Bool;
      _w10 : Bool;
      _w11 : Bool;
      _w12 : Bool;
   END_VAR
BEGIN

REGION Network 1: convertir temporizadores
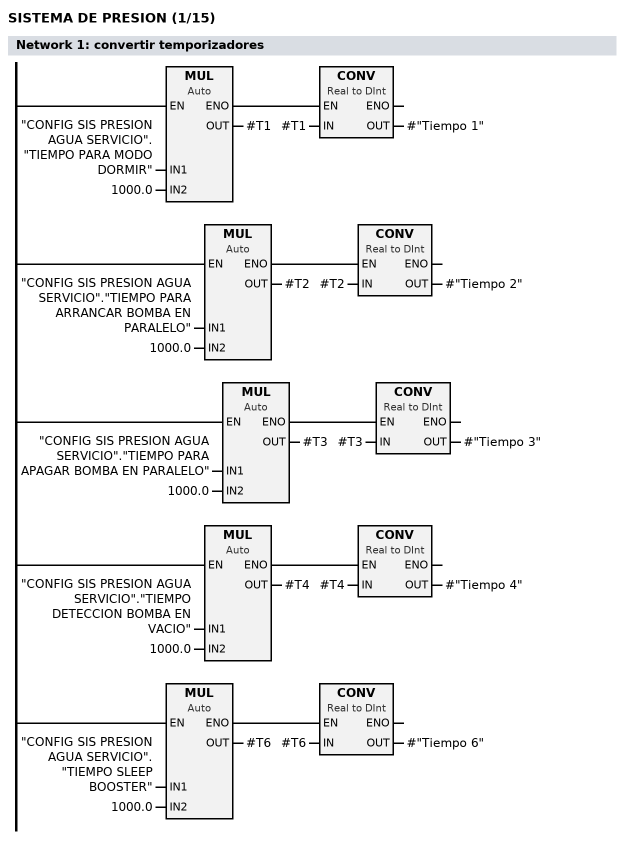
   RUNG wire#powerrail
      Mul(in1 := "CONFIG SIS PRESION AGUA SERVICIO"."TIEMPO PARA MODO DORMIR", in2 := 1000.0, out => #T1)
      { S7_Templates := "[SrcType := Real, DestType := DInt]" } Convert(in := #T1, out => #"Tiempo 1")
   END_RUNG
   RUNG wire#powerrail
      Mul(in1 := "CONFIG SIS PRESION AGUA SERVICIO"."TIEMPO PARA ARRANCAR BOMBA EN PARALELO", in2 := 1000.0, out => #T2)
      { S7_Templates := "[SrcType := Real, DestType := DInt]" } Convert(in := #T2, out => #"Tiempo 2")
   END_RUNG
   RUNG wire#powerrail
      Mul(in1 := "CONFIG SIS PRESION AGUA SERVICIO"."TIEMPO PARA APAGAR BOMBA EN PARALELO", in2 := 1000.0, out => #T3)
      { S7_Templates := "[SrcType := Real, DestType := DInt]" } Convert(in := #T3, out => #"Tiempo 3")
   END_RUNG
   RUNG wire#powerrail
      Mul(in1 := "CONFIG SIS PRESION AGUA SERVICIO"."TIEMPO DETECCION BOMBA EN VACIO", in2 := 1000.0, out => #T4)
      { S7_Templates := "[SrcType := Real, DestType := DInt]" } Convert(in := #T4, out => #"Tiempo 4")
   END_RUNG
   RUNG wire#powerrail
      Mul(in1 := "CONFIG SIS PRESION AGUA SERVICIO"."TIEMPO SLEEP BOOSTER", in2 := 1000.0, out => #T6)
      { S7_Templates := "[SrcType := Real, DestType := DInt]" } Convert(in := #T6, out => #"Tiempo 6")
   END_RUNG
   // the same network as SCL:
   #T1 := "CONFIG SIS PRESION AGUA SERVICIO"."TIEMPO PARA MODO DORMIR" * 1000.0;
   #"Tiempo 1" := REAL_TO_DINT(#T1);
   #T2 := "CONFIG SIS PRESION AGUA SERVICIO"."TIEMPO PARA ARRANCAR BOMBA EN PARALELO" * 1000.0;
   #"Tiempo 2" := REAL_TO_DINT(#T2);
   #T3 := "CONFIG SIS PRESION AGUA SERVICIO"."TIEMPO PARA APAGAR BOMBA EN PARALELO" * 1000.0;
   #"Tiempo 3" := REAL_TO_DINT(#T3);
   #T4 := "CONFIG SIS PRESION AGUA SERVICIO"."TIEMPO DETECCION BOMBA EN VACIO" * 1000.0;
   #"Tiempo 4" := REAL_TO_DINT(#T4);
   #T6 := "CONFIG SIS PRESION AGUA SERVICIO"."TIEMPO SLEEP BOOSTER" * 1000.0;
   #"Tiempo 6" := REAL_TO_DINT(#T6);
END_REGION

REGION Network 2: FRECUENCIA DE OPERACION
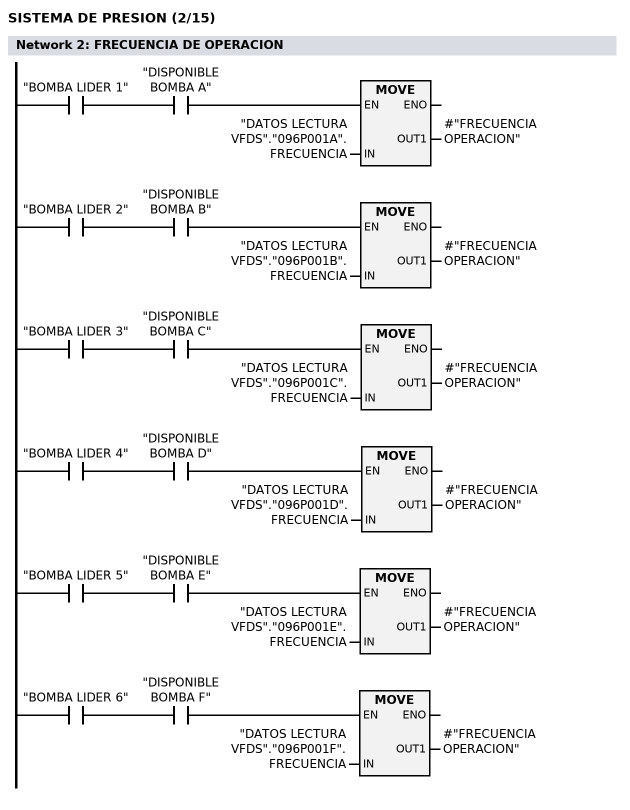
   RUNG wire#powerrail
      Contact( "BOMBA LIDER 1" )
      Contact( "DISPONIBLE BOMBA A" )
      Move(in := "DATOS LECTURA VFDS"."096P001A".FRECUENCIA, out1 => #"FRECUENCIA OPERACION")
   END_RUNG
   RUNG wire#powerrail
      Contact( "BOMBA LIDER 2" )
      Contact( "DISPONIBLE BOMBA B" )
      Move(in := "DATOS LECTURA VFDS"."096P001B".FRECUENCIA, out1 => #"FRECUENCIA OPERACION")
   END_RUNG
   RUNG wire#powerrail
      Contact( "BOMBA LIDER 3" )
      Contact( "DISPONIBLE BOMBA C" )
      Move(in := "DATOS LECTURA VFDS"."096P001C".FRECUENCIA, out1 => #"FRECUENCIA OPERACION")
   END_RUNG
   RUNG wire#powerrail
      Contact( "BOMBA LIDER 4" )
      Contact( "DISPONIBLE BOMBA D" )
      Move(in := "DATOS LECTURA VFDS"."096P001D".FRECUENCIA, out1 => #"FRECUENCIA OPERACION")
   END_RUNG
   RUNG wire#powerrail
      Contact( "BOMBA LIDER 5" )
      Contact( "DISPONIBLE BOMBA E" )
      Move(in := "DATOS LECTURA VFDS"."096P001E".FRECUENCIA, out1 => #"FRECUENCIA OPERACION")
   END_RUNG
   RUNG wire#powerrail
      Contact( "BOMBA LIDER 6" )
      Contact( "DISPONIBLE BOMBA F" )
      Move(in := "DATOS LECTURA VFDS"."096P001F".FRECUENCIA, out1 => #"FRECUENCIA OPERACION")
   END_RUNG
   // the same network as SCL:
   IF "BOMBA LIDER 1" AND "DISPONIBLE BOMBA A" THEN
       #"FRECUENCIA OPERACION" := "DATOS LECTURA VFDS"."096P001A".FRECUENCIA;
   END_IF;
   IF "BOMBA LIDER 2" AND "DISPONIBLE BOMBA B" THEN
       #"FRECUENCIA OPERACION" := "DATOS LECTURA VFDS"."096P001B".FRECUENCIA;
   END_IF;
   IF "BOMBA LIDER 3" AND "DISPONIBLE BOMBA C" THEN
       #"FRECUENCIA OPERACION" := "DATOS LECTURA VFDS"."096P001C".FRECUENCIA;
   END_IF;
   IF "BOMBA LIDER 4" AND "DISPONIBLE BOMBA D" THEN
       #"FRECUENCIA OPERACION" := "DATOS LECTURA VFDS"."096P001D".FRECUENCIA;
   END_IF;
   IF "BOMBA LIDER 5" AND "DISPONIBLE BOMBA E" THEN
       #"FRECUENCIA OPERACION" := "DATOS LECTURA VFDS"."096P001E".FRECUENCIA;
   END_IF;
   IF "BOMBA LIDER 6" AND "DISPONIBLE BOMBA F" THEN
       #"FRECUENCIA OPERACION" := "DATOS LECTURA VFDS"."096P001F".FRECUENCIA;
   END_IF;
END_REGION

REGION Network 3: DORMIR DESPERTAR
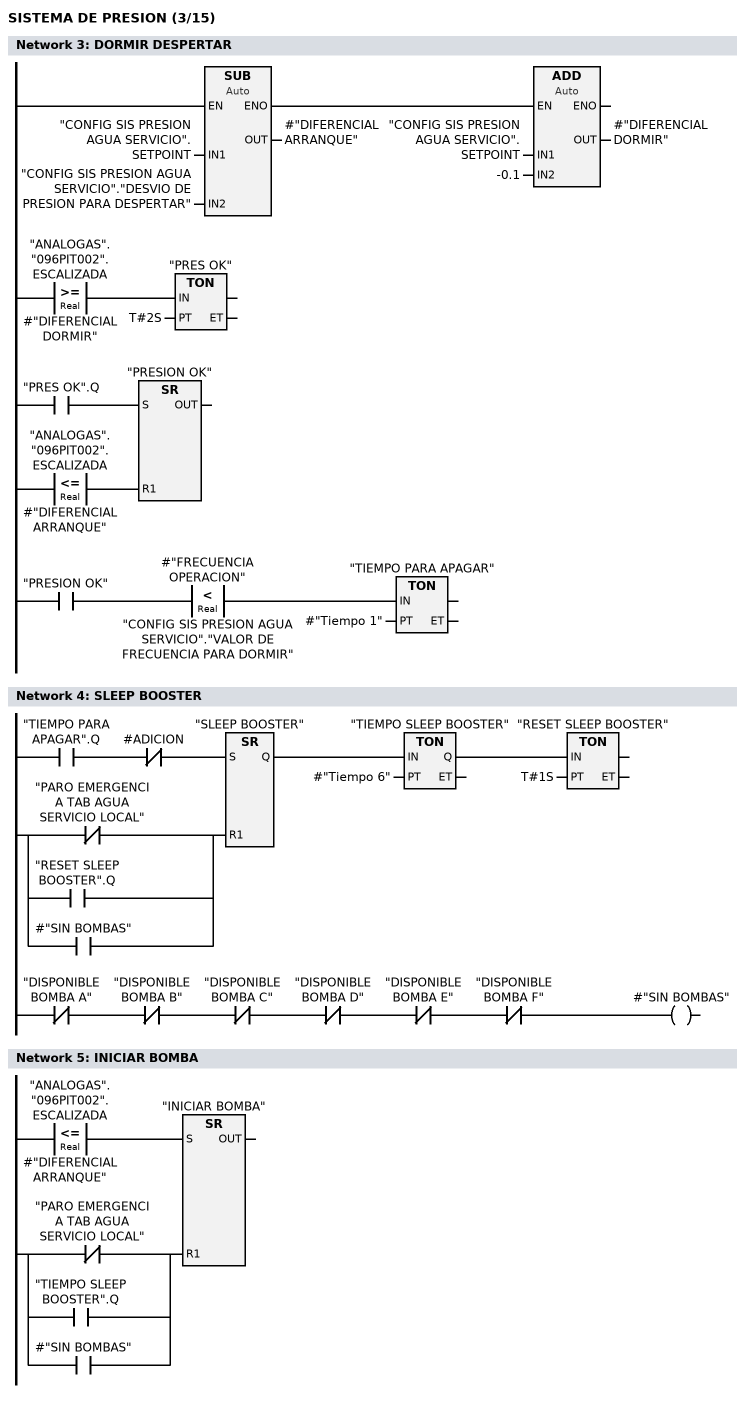
   #"DIFERENCIAL ARRANQUE" := "CONFIG SIS PRESION AGUA SERVICIO".SETPOINT - "CONFIG SIS PRESION AGUA SERVICIO"."DESVIO DE PRESION PARA DESPERTAR";
   #"DIFERENCIAL DORMIR" := "CONFIG SIS PRESION AGUA SERVICIO".SETPOINT + (-0.1);
   "PRES OK".TON(IN := "ANALOGAS"."096PIT002".ESCALIZADA >= #"DIFERENCIAL DORMIR", PT := T#2S);
   IF "PRES OK".Q THEN
       "PRESION OK" := TRUE;   // SR flip-flop
   END_IF;
   IF "ANALOGAS"."096PIT002".ESCALIZADA <= #"DIFERENCIAL ARRANQUE" THEN "PRESION OK" := FALSE; END_IF;
   "TIEMPO PARA APAGAR".TON(IN := "PRESION OK" AND (#"FRECUENCIA OPERACION" < "CONFIG SIS PRESION AGUA SERVICIO"."VALOR DE FRECUENCIA PARA DORMIR"),
                           PT := #"Tiempo 1");
END_REGION

REGION Network 4: SLEEP BOOSTER
   IF "TIEMPO PARA APAGAR".Q AND NOT #ADICION THEN
       "SLEEP BOOSTER" := TRUE;   // SR flip-flop
   END_IF;
   IF NOT "PARO EMERGENCIA TAB AGUA SERVICIO LOCAL" OR "RESET SLEEP BOOSTER".Q OR #"SIN BOMBAS" THEN
       "SLEEP BOOSTER" := FALSE;
   END_IF;
   "TIEMPO SLEEP BOOSTER".TON(IN := "SLEEP BOOSTER", PT := #"Tiempo 6");
   "RESET SLEEP BOOSTER".TON(IN := "TIEMPO SLEEP BOOSTER".Q, PT := T#1S);
   #"SIN BOMBAS" := NOT "DISPONIBLE BOMBA A" AND NOT "DISPONIBLE BOMBA B" AND NOT "DISPONIBLE BOMBA C" AND NOT "DISPONIBLE BOMBA D" AND NOT "DISPONIBLE BOMBA E" AND NOT "DISPONIBLE BOMBA F";
END_REGION

REGION Network 5: INICIAR BOMBA
   RUNG wire#powerrail
      { S7_Templates := "SrcType := Real" } LE_Contact(in1 := "ANALOGAS"."096PIT002".ESCALIZADA, in2 := #"DIFERENCIAL ARRANQUE")
      S_SR(operand := "INICIAR BOMBA", r1 := wire#w1)
   END_RUNG
   RUNG wire#powerrail
      I_Contact( "PARO EMERGENCIA TAB AGUA SERVICIO LOCAL" )
   END_RUNG wire#w1
   RUNG wire#powerrail
      Contact( "TIEMPO SLEEP BOOSTER".Q )
   END_RUNG wire#w1
   RUNG wire#powerrail
      Contact( #"SIN BOMBAS" )
   END_RUNG wire#w1
   // the same network as SCL:
   IF "ANALOGAS"."096PIT002".ESCALIZADA <= #"DIFERENCIAL ARRANQUE" THEN
       "INICIAR BOMBA" := TRUE;   // SR flip-flop
   END_IF;
   IF NOT "PARO EMERGENCIA TAB AGUA SERVICIO LOCAL" OR "TIEMPO SLEEP BOOSTER".Q OR #"SIN BOMBAS" THEN
       "INICIAR BOMBA" := FALSE;
   END_IF;
END_REGION

REGION Network 6: CONTEO BOMBA A
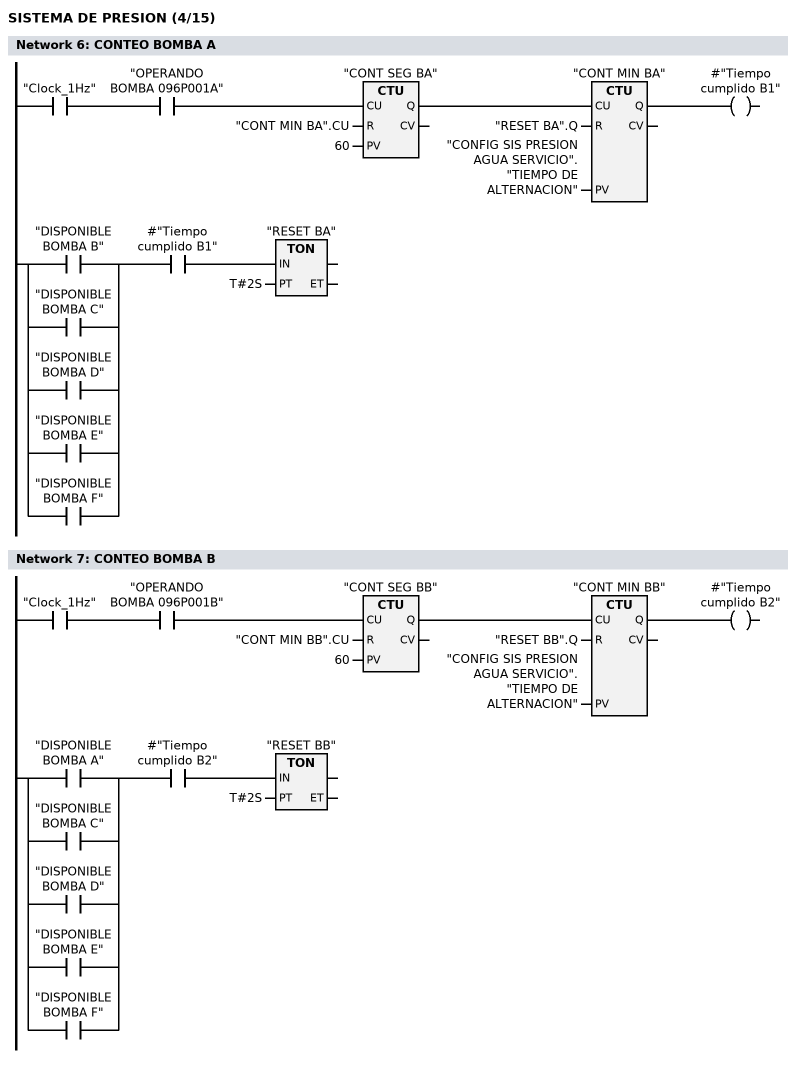
   "CONT SEG BA".CTU(CU := "Clock_1Hz" AND "OPERANDO BOMBA 096P001A", R := "CONT MIN BA".CU, PV := 60);
   "CONT MIN BA".CTU(CU := "CONT SEG BA".Q,
                     R := "RESET BA".Q,
                     PV := "CONFIG SIS PRESION AGUA SERVICIO"."TIEMPO DE ALTERNACION");
   #"Tiempo cumplido B1" := "CONT MIN BA".Q;
   "RESET BA".TON(IN := ("DISPONIBLE BOMBA B" OR "DISPONIBLE BOMBA C" OR "DISPONIBLE BOMBA D" OR "DISPONIBLE BOMBA E" OR "DISPONIBLE BOMBA F") AND #"Tiempo cumplido B1",
                  PT := T#2S);
END_REGION

REGION Network 7: CONTEO BOMBA B
   "CONT SEG BB".CTU(CU := "Clock_1Hz" AND "OPERANDO BOMBA 096P001B", R := "CONT MIN BB".CU, PV := 60);
   "CONT MIN BB".CTU(CU := "CONT SEG BB".Q,
                     R := "RESET BB".Q,
                     PV := "CONFIG SIS PRESION AGUA SERVICIO"."TIEMPO DE ALTERNACION");
   #"Tiempo cumplido B2" := "CONT MIN BB".Q;
   "RESET BB".TON(IN := ("DISPONIBLE BOMBA A" OR "DISPONIBLE BOMBA C" OR "DISPONIBLE BOMBA D" OR "DISPONIBLE BOMBA E" OR "DISPONIBLE BOMBA F") AND #"Tiempo cumplido B2",
                  PT := T#2S);
END_REGION

REGION Network 8: CONTEO BOMBA C
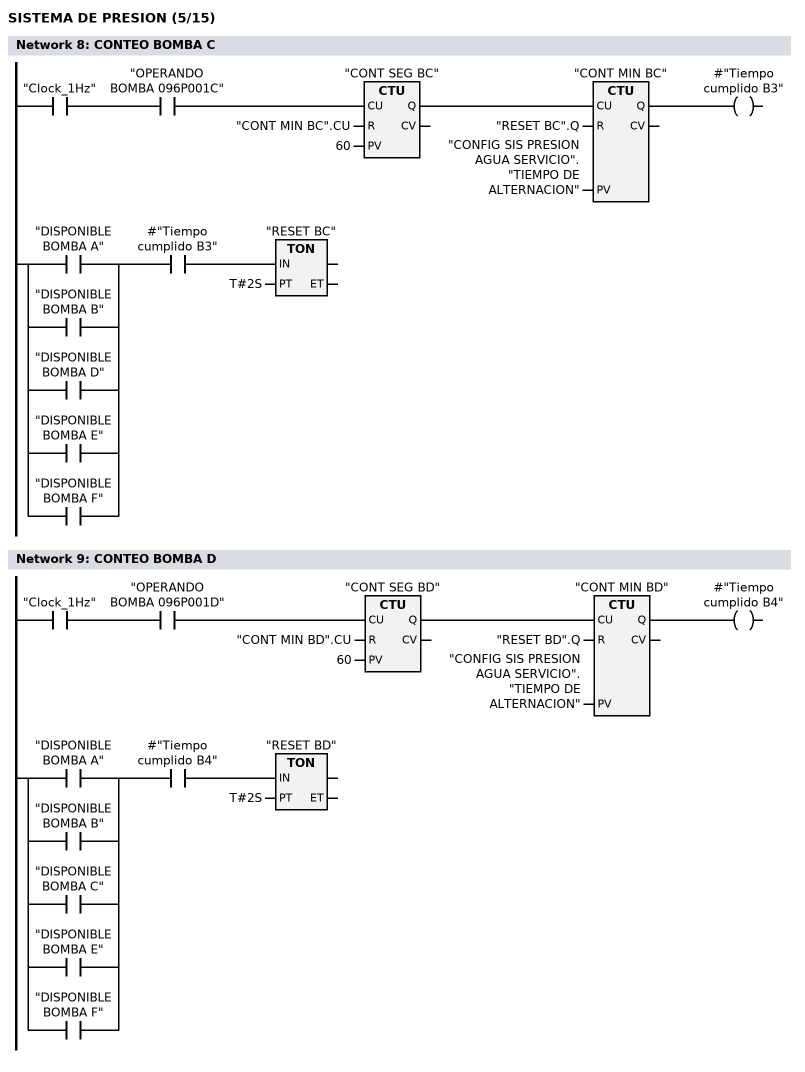
   "CONT SEG BC".CTU(CU := "Clock_1Hz" AND "OPERANDO BOMBA 096P001C", R := "CONT MIN BC".CU, PV := 60);
   "CONT MIN BC".CTU(CU := "CONT SEG BC".Q,
                     R := "RESET BC".Q,
                     PV := "CONFIG SIS PRESION AGUA SERVICIO"."TIEMPO DE ALTERNACION");
   #"Tiempo cumplido B3" := "CONT MIN BC".Q;
   "RESET BC".TON(IN := ("DISPONIBLE BOMBA A" OR "DISPONIBLE BOMBA B" OR "DISPONIBLE BOMBA D" OR "DISPONIBLE BOMBA E" OR "DISPONIBLE BOMBA F") AND #"Tiempo cumplido B3",
                  PT := T#2S);
END_REGION

REGION Network 9: CONTEO BOMBA D
   "CONT SEG BD".CTU(CU := "Clock_1Hz" AND "OPERANDO BOMBA 096P001D", R := "CONT MIN BD".CU, PV := 60);
   "CONT MIN BD".CTU(CU := "CONT SEG BD".Q,
                     R := "RESET BD".Q,
                     PV := "CONFIG SIS PRESION AGUA SERVICIO"."TIEMPO DE ALTERNACION");
   #"Tiempo cumplido B4" := "CONT MIN BD".Q;
   "RESET BD".TON(IN := ("DISPONIBLE BOMBA A" OR "DISPONIBLE BOMBA B" OR "DISPONIBLE BOMBA C" OR "DISPONIBLE BOMBA E" OR "DISPONIBLE BOMBA F") AND #"Tiempo cumplido B4",
                  PT := T#2S);
END_REGION

REGION Network 10: CONTEO BOMBA E
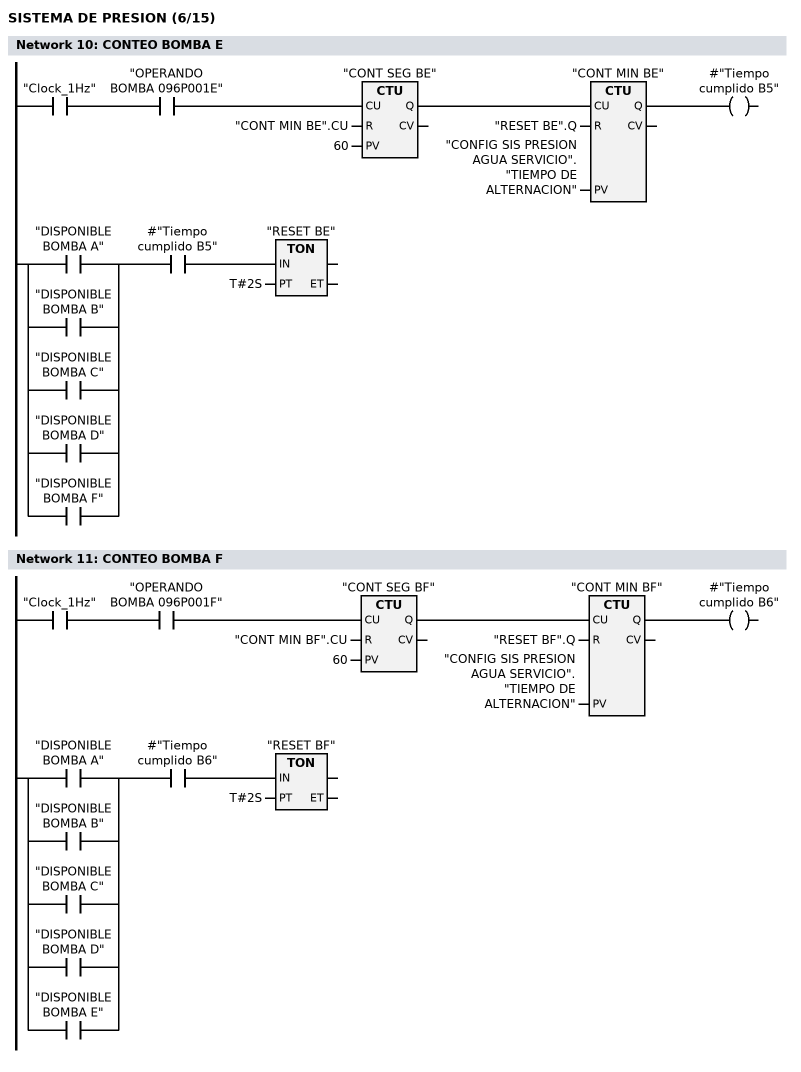
   "CONT SEG BE".CTU(CU := "Clock_1Hz" AND "OPERANDO BOMBA 096P001E", R := "CONT MIN BE".CU, PV := 60);
   "CONT MIN BE".CTU(CU := "CONT SEG BE".Q,
                     R := "RESET BE".Q,
                     PV := "CONFIG SIS PRESION AGUA SERVICIO"."TIEMPO DE ALTERNACION");
   #"Tiempo cumplido B5" := "CONT MIN BE".Q;
   "RESET BE".TON(IN := ("DISPONIBLE BOMBA A" OR "DISPONIBLE BOMBA B" OR "DISPONIBLE BOMBA C" OR "DISPONIBLE BOMBA D" OR "DISPONIBLE BOMBA F") AND #"Tiempo cumplido B5",
                  PT := T#2S);
END_REGION

REGION Network 11: CONTEO BOMBA F
   "CONT SEG BF".CTU(CU := "Clock_1Hz" AND "OPERANDO BOMBA 096P001F", R := "CONT MIN BF".CU, PV := 60);
   "CONT MIN BF".CTU(CU := "CONT SEG BF".Q,
                     R := "RESET BF".Q,
                     PV := "CONFIG SIS PRESION AGUA SERVICIO"."TIEMPO DE ALTERNACION");
   #"Tiempo cumplido B6" := "CONT MIN BF".Q;
   "RESET BF".TON(IN := ("DISPONIBLE BOMBA A" OR "DISPONIBLE BOMBA B" OR "DISPONIBLE BOMBA C" OR "DISPONIBLE BOMBA D" OR "DISPONIBLE BOMBA E") AND #"Tiempo cumplido B6",
                  PT := T#2S);
END_REGION

REGION Network 12: CONTADOR ALTERNACION
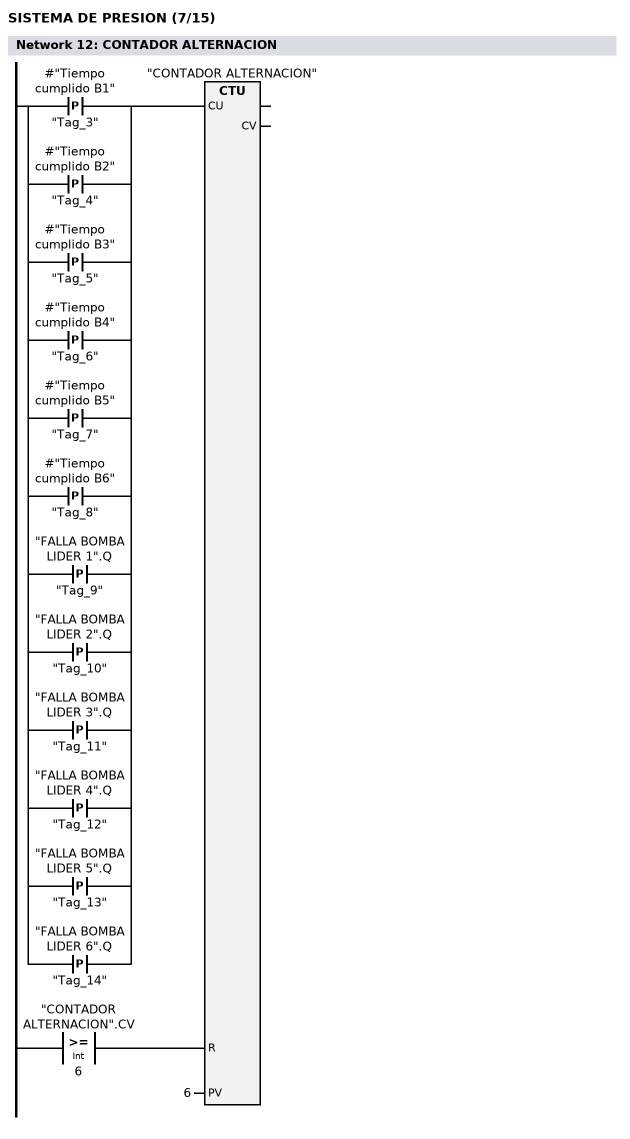
   #_w1 := #"Tiempo cumplido B1" AND NOT "Tag_3";   // rising edge of #"Tiempo cumplido B1"
   "Tag_3" := #"Tiempo cumplido B1";
   #_w2 := #"Tiempo cumplido B2" AND NOT "Tag_4";   // rising edge of #"Tiempo cumplido B2"
   "Tag_4" := #"Tiempo cumplido B2";
   #_w3 := #"Tiempo cumplido B3" AND NOT "Tag_5";   // rising edge of #"Tiempo cumplido B3"
   "Tag_5" := #"Tiempo cumplido B3";
   #_w4 := #"Tiempo cumplido B4" AND NOT "Tag_6";   // rising edge of #"Tiempo cumplido B4"
   "Tag_6" := #"Tiempo cumplido B4";
   #_w5 := #"Tiempo cumplido B5" AND NOT "Tag_7";   // rising edge of #"Tiempo cumplido B5"
   "Tag_7" := #"Tiempo cumplido B5";
   #_w6 := #"Tiempo cumplido B6" AND NOT "Tag_8";   // rising edge of #"Tiempo cumplido B6"
   "Tag_8" := #"Tiempo cumplido B6";
   #_w7 := "FALLA BOMBA LIDER 1".Q AND NOT "Tag_9";   // rising edge of "FALLA BOMBA LIDER 1".Q
   "Tag_9" := "FALLA BOMBA LIDER 1".Q;
   #_w8 := "FALLA BOMBA LIDER 2".Q AND NOT "Tag_10";   // rising edge of "FALLA BOMBA LIDER 2".Q
   "Tag_10" := "FALLA BOMBA LIDER 2".Q;
   #_w9 := "FALLA BOMBA LIDER 3".Q AND NOT "Tag_11";   // rising edge of "FALLA BOMBA LIDER 3".Q
   "Tag_11" := "FALLA BOMBA LIDER 3".Q;
   #_w10 := "FALLA BOMBA LIDER 4".Q AND NOT "Tag_12";   // rising edge of "FALLA BOMBA LIDER 4".Q
   "Tag_12" := "FALLA BOMBA LIDER 4".Q;
   #_w11 := "FALLA BOMBA LIDER 5".Q AND NOT "Tag_13";   // rising edge of "FALLA BOMBA LIDER 5".Q
   "Tag_13" := "FALLA BOMBA LIDER 5".Q;
   #_w12 := "FALLA BOMBA LIDER 6".Q AND NOT "Tag_14";   // rising edge of "FALLA BOMBA LIDER 6".Q
   "Tag_14" := "FALLA BOMBA LIDER 6".Q;
   "CONTADOR ALTERNACION".CTU(CU := #_w1 OR #_w2 OR #_w3 OR #_w4 OR #_w5 OR #_w6 OR #_w7 OR #_w8 OR #_w9 OR #_w10 OR #_w11 OR #_w12,
                           R := "CONTADOR ALTERNACION".CV >= 6,
                           PV := 6);
END_REGION

REGION Network 13: FALLA BOMBA LIDER
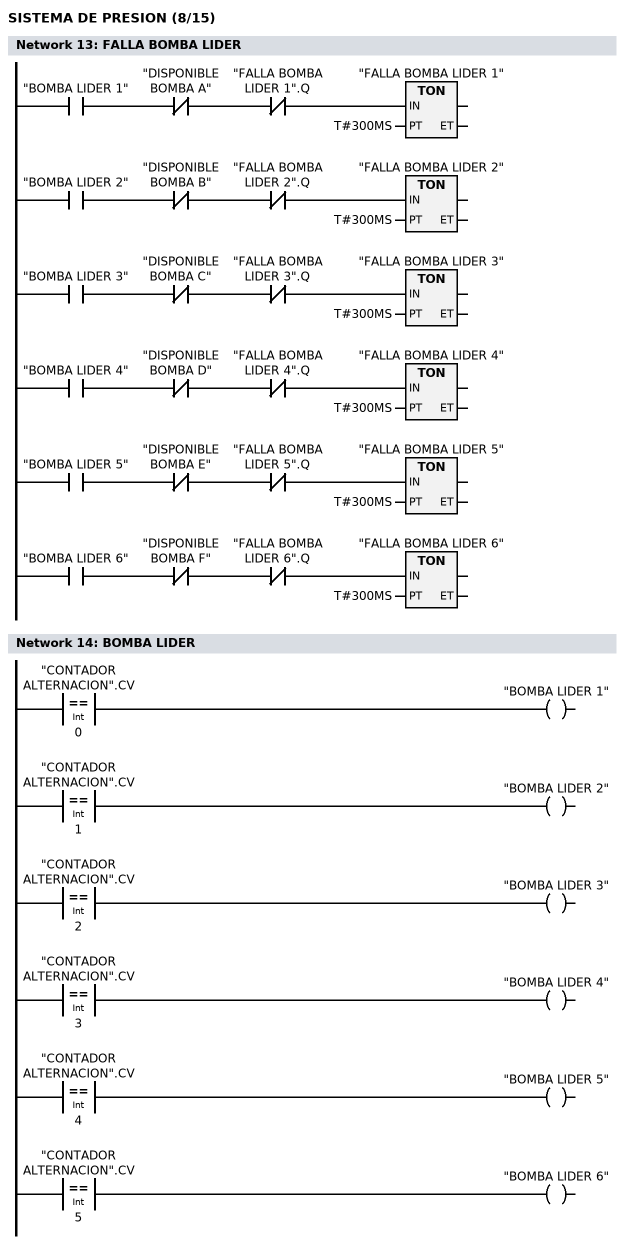
   "FALLA BOMBA LIDER 1".TON(IN := "BOMBA LIDER 1" AND NOT "DISPONIBLE BOMBA A" AND NOT "FALLA BOMBA LIDER 1".Q,
                           PT := T#300MS);
   "FALLA BOMBA LIDER 2".TON(IN := "BOMBA LIDER 2" AND NOT "DISPONIBLE BOMBA B" AND NOT "FALLA BOMBA LIDER 2".Q,
                           PT := T#300MS);
   "FALLA BOMBA LIDER 3".TON(IN := "BOMBA LIDER 3" AND NOT "DISPONIBLE BOMBA C" AND NOT "FALLA BOMBA LIDER 3".Q,
                           PT := T#300MS);
   "FALLA BOMBA LIDER 4".TON(IN := "BOMBA LIDER 4" AND NOT "DISPONIBLE BOMBA D" AND NOT "FALLA BOMBA LIDER 4".Q,
                           PT := T#300MS);
   "FALLA BOMBA LIDER 5".TON(IN := "BOMBA LIDER 5" AND NOT "DISPONIBLE BOMBA E" AND NOT "FALLA BOMBA LIDER 5".Q,
                           PT := T#300MS);
   "FALLA BOMBA LIDER 6".TON(IN := "BOMBA LIDER 6" AND NOT "DISPONIBLE BOMBA F" AND NOT "FALLA BOMBA LIDER 6".Q,
                           PT := T#300MS);
END_REGION

REGION Network 14: BOMBA LIDER
   RUNG wire#powerrail
      { S7_Templates := "SrcType := Int" } EQ_Contact(in1 := "CONTADOR ALTERNACION".CV, in2 := 0)
      Coil( "BOMBA LIDER 1" )
   END_RUNG
   RUNG wire#powerrail
      { S7_Templates := "SrcType := Int" } EQ_Contact(in1 := "CONTADOR ALTERNACION".CV, in2 := 1)
      Coil( "BOMBA LIDER 2" )
   END_RUNG
   RUNG wire#powerrail
      { S7_Templates := "SrcType := Int" } EQ_Contact(in1 := "CONTADOR ALTERNACION".CV, in2 := 2)
      Coil( "BOMBA LIDER 3" )
   END_RUNG
   RUNG wire#powerrail
      { S7_Templates := "SrcType := Int" } EQ_Contact(in1 := "CONTADOR ALTERNACION".CV, in2 := 3)
      Coil( "BOMBA LIDER 4" )
   END_RUNG
   RUNG wire#powerrail
      { S7_Templates := "SrcType := Int" } EQ_Contact(in1 := "CONTADOR ALTERNACION".CV, in2 := 4)
      Coil( "BOMBA LIDER 5" )
   END_RUNG
   RUNG wire#powerrail
      { S7_Templates := "SrcType := Int" } EQ_Contact(in1 := "CONTADOR ALTERNACION".CV, in2 := 5)
      Coil( "BOMBA LIDER 6" )
   END_RUNG
   // the same network as SCL:
   "BOMBA LIDER 1" := "CONTADOR ALTERNACION".CV = 0;
   "BOMBA LIDER 2" := "CONTADOR ALTERNACION".CV = 1;
   "BOMBA LIDER 3" := "CONTADOR ALTERNACION".CV = 2;
   "BOMBA LIDER 4" := "CONTADOR ALTERNACION".CV = 3;
   "BOMBA LIDER 5" := "CONTADOR ALTERNACION".CV = 4;
   "BOMBA LIDER 6" := "CONTADOR ALTERNACION".CV = 5;
END_REGION

REGION Network 15: ADICION
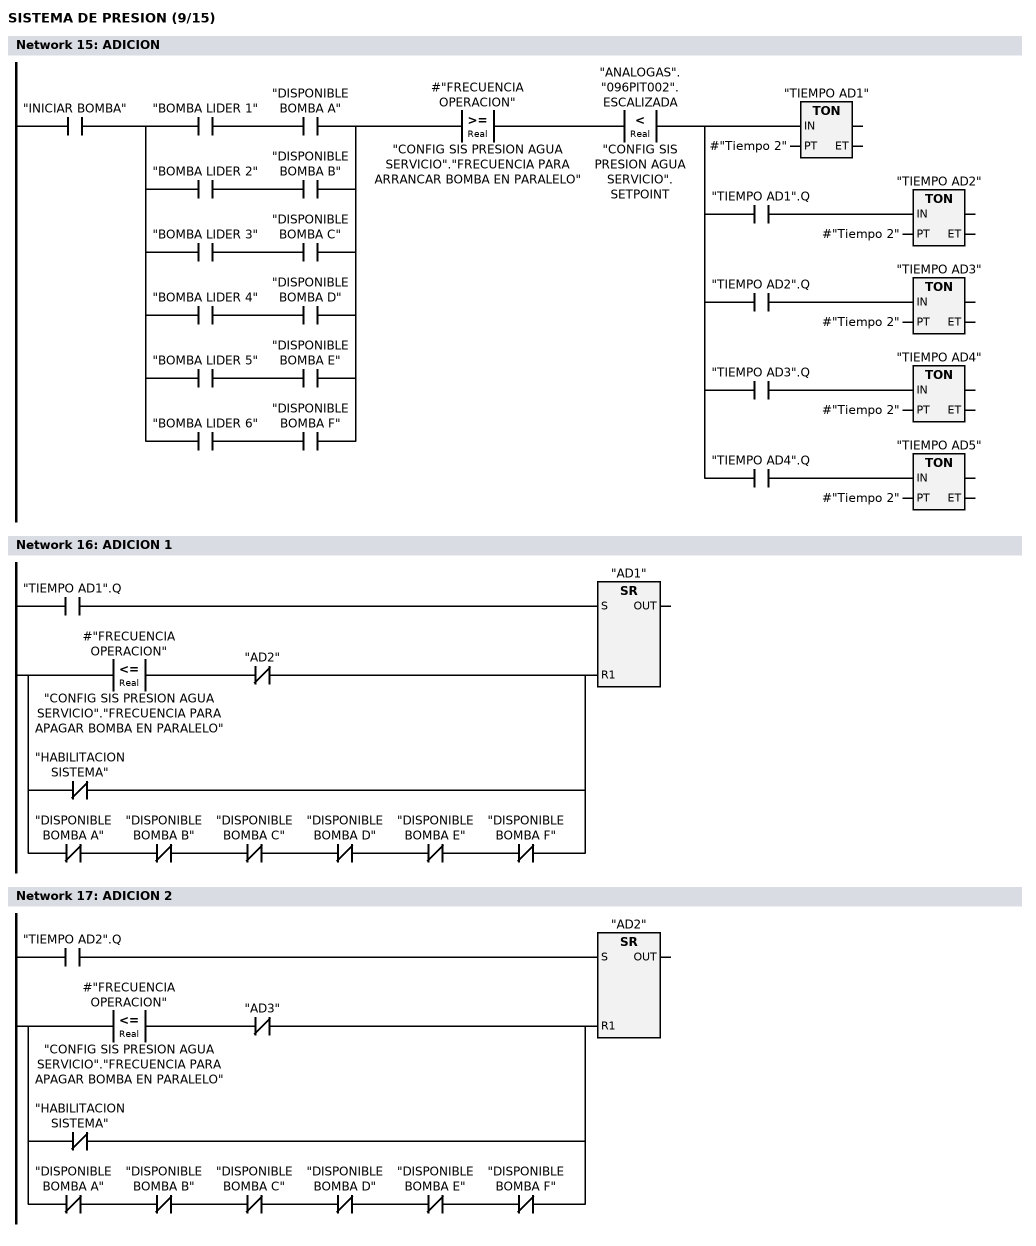
   #_w1 := "INICIAR BOMBA" AND (("BOMBA LIDER 1" AND "DISPONIBLE BOMBA A") OR ("BOMBA LIDER 2" AND "DISPONIBLE BOMBA B") OR ("BOMBA LIDER 3" AND "DISPONIBLE BOMBA C") OR ("BOMBA LIDER 4" AND "DISPONIBLE BOMBA D") OR ("BOMBA LIDER 5" AND "DISPONIBLE BOMBA E") OR ("BOMBA LIDER 6" AND "DISPONIBLE BOMBA F")) AND (#"FRECUENCIA OPERACION" >= "CONFIG SIS PRESION AGUA SERVICIO"."FRECUENCIA PARA ARRANCAR BOMBA EN PARALELO") AND ("ANALOGAS"."096PIT002".ESCALIZADA < "CONFIG SIS PRESION AGUA SERVICIO".SETPOINT);
   "TIEMPO AD1".TON(IN := #_w1, PT := #"Tiempo 2");
   "TIEMPO AD2".TON(IN := #_w1 AND "TIEMPO AD1".Q, PT := #"Tiempo 2");
   "TIEMPO AD3".TON(IN := #_w1 AND "TIEMPO AD2".Q, PT := #"Tiempo 2");
   "TIEMPO AD4".TON(IN := #_w1 AND "TIEMPO AD3".Q, PT := #"Tiempo 2");
   "TIEMPO AD5".TON(IN := #_w1 AND "TIEMPO AD4".Q, PT := #"Tiempo 2");
END_REGION

REGION Network 16: ADICION 1
   RUNG wire#powerrail
      Contact( "TIEMPO AD1".Q )
      S_SR(operand := "AD1", r1 := wire#w1)
   END_RUNG
   RUNG wire#powerrail
      { S7_Templates := "SrcType := Real" } LE_Contact(in1 := #"FRECUENCIA OPERACION", in2 := "CONFIG SIS PRESION AGUA SERVICIO"."FRECUENCIA PARA APAGAR BOMBA EN PARALELO")
      I_Contact( "AD2" )
   END_RUNG wire#w1
   RUNG wire#powerrail
      I_Contact( "HABILITACION SISTEMA" )
   END_RUNG wire#w1
   RUNG wire#powerrail
      I_Contact( "DISPONIBLE BOMBA A" )
      I_Contact( "DISPONIBLE BOMBA B" )
      I_Contact( "DISPONIBLE BOMBA C" )
      I_Contact( "DISPONIBLE BOMBA D" )
      I_Contact( "DISPONIBLE BOMBA E" )
      I_Contact( "DISPONIBLE BOMBA F" )
   END_RUNG wire#w1
   // the same network as SCL:
   IF "TIEMPO AD1".Q THEN
       "AD1" := TRUE;   // SR flip-flop
   END_IF;
   IF ((#"FRECUENCIA OPERACION" <= "CONFIG SIS PRESION AGUA SERVICIO"."FRECUENCIA PARA APAGAR BOMBA EN PARALELO") AND NOT "AD2") OR NOT "HABILITACION SISTEMA" OR (NOT "DISPONIBLE BOMBA A" AND NOT "DISPONIBLE BOMBA B" AND NOT "DISPONIBLE BOMBA C" AND NOT "DISPONIBLE BOMBA D" AND NOT "DISPONIBLE BOMBA E" AND NOT "DISPONIBLE BOMBA F") THEN
       "AD1" := FALSE;
   END_IF;
END_REGION

REGION Network 17: ADICION 2
   RUNG wire#powerrail
      Contact( "TIEMPO AD2".Q )
      S_SR(operand := "AD2", r1 := wire#w1)
   END_RUNG
   RUNG wire#powerrail
      { S7_Templates := "SrcType := Real" } LE_Contact(in1 := #"FRECUENCIA OPERACION", in2 := "CONFIG SIS PRESION AGUA SERVICIO"."FRECUENCIA PARA APAGAR BOMBA EN PARALELO")
      I_Contact( "AD3" )
   END_RUNG wire#w1
   RUNG wire#powerrail
      I_Contact( "HABILITACION SISTEMA" )
   END_RUNG wire#w1
   RUNG wire#powerrail
      I_Contact( "DISPONIBLE BOMBA A" )
      I_Contact( "DISPONIBLE BOMBA B" )
      I_Contact( "DISPONIBLE BOMBA C" )
      I_Contact( "DISPONIBLE BOMBA D" )
      I_Contact( "DISPONIBLE BOMBA E" )
      I_Contact( "DISPONIBLE BOMBA F" )
   END_RUNG wire#w1
   // the same network as SCL:
   IF "TIEMPO AD2".Q THEN
       "AD2" := TRUE;   // SR flip-flop
   END_IF;
   IF ((#"FRECUENCIA OPERACION" <= "CONFIG SIS PRESION AGUA SERVICIO"."FRECUENCIA PARA APAGAR BOMBA EN PARALELO") AND NOT "AD3") OR NOT "HABILITACION SISTEMA" OR (NOT "DISPONIBLE BOMBA A" AND NOT "DISPONIBLE BOMBA B" AND NOT "DISPONIBLE BOMBA C" AND NOT "DISPONIBLE BOMBA D" AND NOT "DISPONIBLE BOMBA E" AND NOT "DISPONIBLE BOMBA F") THEN
       "AD2" := FALSE;
   END_IF;
END_REGION

REGION Network 18: ADICION 3
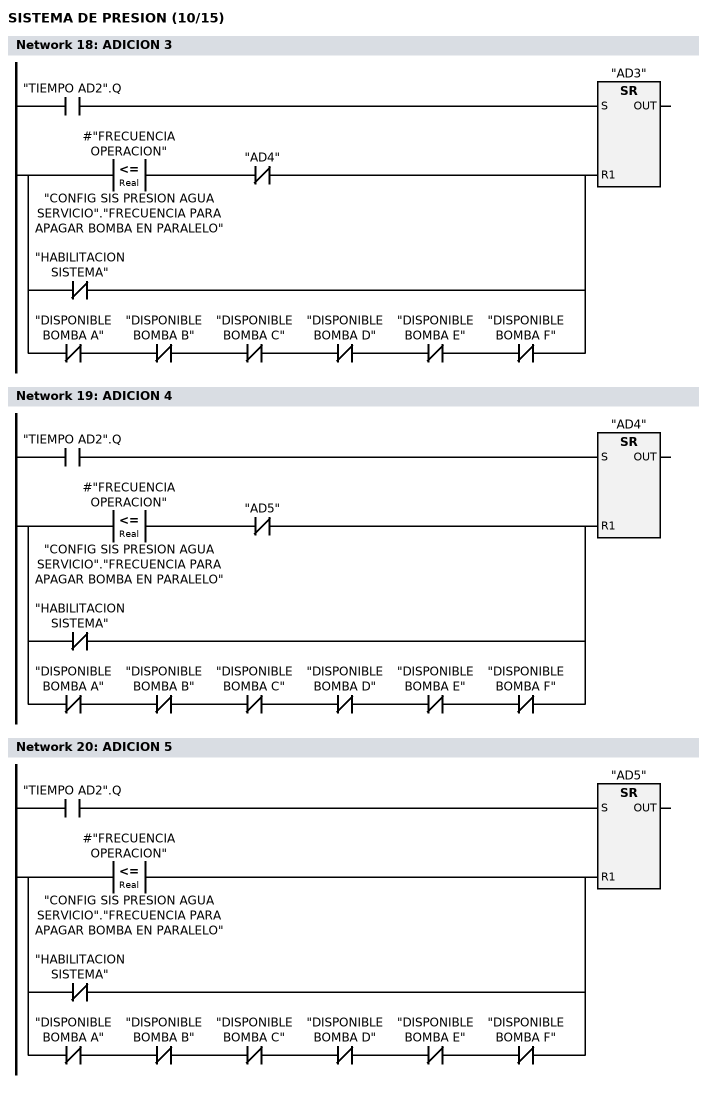
   RUNG wire#powerrail
      Contact( "TIEMPO AD2".Q )
      S_SR(operand := "AD3", r1 := wire#w1)
   END_RUNG
   RUNG wire#powerrail
      { S7_Templates := "SrcType := Real" } LE_Contact(in1 := #"FRECUENCIA OPERACION", in2 := "CONFIG SIS PRESION AGUA SERVICIO"."FRECUENCIA PARA APAGAR BOMBA EN PARALELO")
      I_Contact( "AD4" )
   END_RUNG wire#w1
   RUNG wire#powerrail
      I_Contact( "HABILITACION SISTEMA" )
   END_RUNG wire#w1
   RUNG wire#powerrail
      I_Contact( "DISPONIBLE BOMBA A" )
      I_Contact( "DISPONIBLE BOMBA B" )
      I_Contact( "DISPONIBLE BOMBA C" )
      I_Contact( "DISPONIBLE BOMBA D" )
      I_Contact( "DISPONIBLE BOMBA E" )
      I_Contact( "DISPONIBLE BOMBA F" )
   END_RUNG wire#w1
   // the same network as SCL:
   IF "TIEMPO AD2".Q THEN
       "AD3" := TRUE;   // SR flip-flop
   END_IF;
   IF ((#"FRECUENCIA OPERACION" <= "CONFIG SIS PRESION AGUA SERVICIO"."FRECUENCIA PARA APAGAR BOMBA EN PARALELO") AND NOT "AD4") OR NOT "HABILITACION SISTEMA" OR (NOT "DISPONIBLE BOMBA A" AND NOT "DISPONIBLE BOMBA B" AND NOT "DISPONIBLE BOMBA C" AND NOT "DISPONIBLE BOMBA D" AND NOT "DISPONIBLE BOMBA E" AND NOT "DISPONIBLE BOMBA F") THEN
       "AD3" := FALSE;
   END_IF;
END_REGION

REGION Network 19: ADICION 4
   RUNG wire#powerrail
      Contact( "TIEMPO AD2".Q )
      S_SR(operand := "AD4", r1 := wire#w1)
   END_RUNG
   RUNG wire#powerrail
      { S7_Templates := "SrcType := Real" } LE_Contact(in1 := #"FRECUENCIA OPERACION", in2 := "CONFIG SIS PRESION AGUA SERVICIO"."FRECUENCIA PARA APAGAR BOMBA EN PARALELO")
      I_Contact( "AD5" )
   END_RUNG wire#w1
   RUNG wire#powerrail
      I_Contact( "HABILITACION SISTEMA" )
   END_RUNG wire#w1
   RUNG wire#powerrail
      I_Contact( "DISPONIBLE BOMBA A" )
      I_Contact( "DISPONIBLE BOMBA B" )
      I_Contact( "DISPONIBLE BOMBA C" )
      I_Contact( "DISPONIBLE BOMBA D" )
      I_Contact( "DISPONIBLE BOMBA E" )
      I_Contact( "DISPONIBLE BOMBA F" )
   END_RUNG wire#w1
   // the same network as SCL:
   IF "TIEMPO AD2".Q THEN
       "AD4" := TRUE;   // SR flip-flop
   END_IF;
   IF ((#"FRECUENCIA OPERACION" <= "CONFIG SIS PRESION AGUA SERVICIO"."FRECUENCIA PARA APAGAR BOMBA EN PARALELO") AND NOT "AD5") OR NOT "HABILITACION SISTEMA" OR (NOT "DISPONIBLE BOMBA A" AND NOT "DISPONIBLE BOMBA B" AND NOT "DISPONIBLE BOMBA C" AND NOT "DISPONIBLE BOMBA D" AND NOT "DISPONIBLE BOMBA E" AND NOT "DISPONIBLE BOMBA F") THEN
       "AD4" := FALSE;
   END_IF;
END_REGION

REGION Network 20: ADICION 5
   RUNG wire#powerrail
      Contact( "TIEMPO AD2".Q )
      S_SR(operand := "AD5", r1 := wire#w1)
   END_RUNG
   RUNG wire#powerrail
      { S7_Templates := "SrcType := Real" } LE_Contact(in1 := #"FRECUENCIA OPERACION", in2 := "CONFIG SIS PRESION AGUA SERVICIO"."FRECUENCIA PARA APAGAR BOMBA EN PARALELO")
   END_RUNG wire#w1
   RUNG wire#powerrail
      I_Contact( "HABILITACION SISTEMA" )
   END_RUNG wire#w1
   RUNG wire#powerrail
      I_Contact( "DISPONIBLE BOMBA A" )
      I_Contact( "DISPONIBLE BOMBA B" )
      I_Contact( "DISPONIBLE BOMBA C" )
      I_Contact( "DISPONIBLE BOMBA D" )
      I_Contact( "DISPONIBLE BOMBA E" )
      I_Contact( "DISPONIBLE BOMBA F" )
   END_RUNG wire#w1
   // the same network as SCL:
   IF "TIEMPO AD2".Q THEN
       "AD5" := TRUE;   // SR flip-flop
   END_IF;
   IF (#"FRECUENCIA OPERACION" <= "CONFIG SIS PRESION AGUA SERVICIO"."FRECUENCIA PARA APAGAR BOMBA EN PARALELO") OR NOT "HABILITACION SISTEMA" OR (NOT "DISPONIBLE BOMBA A" AND NOT "DISPONIBLE BOMBA B" AND NOT "DISPONIBLE BOMBA C" AND NOT "DISPONIBLE BOMBA D" AND NOT "DISPONIBLE BOMBA E" AND NOT "DISPONIBLE BOMBA F") THEN
       "AD5" := FALSE;
   END_IF;
END_REGION

REGION Network 21: ARRANQUE B1
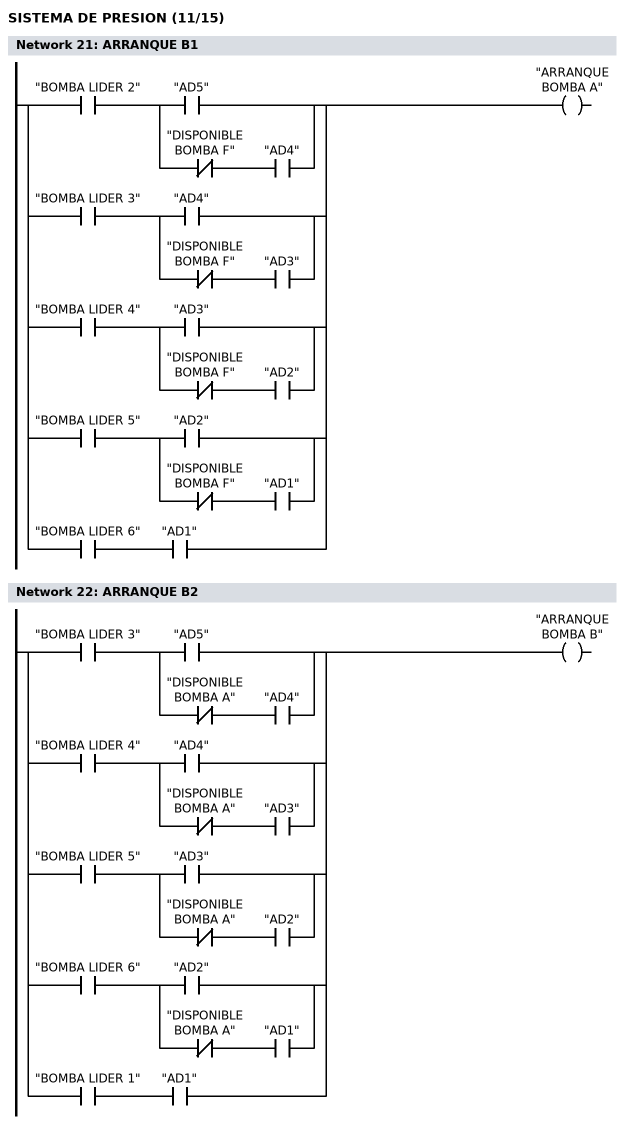
   RUNG wire#powerrail
      Contact( "BOMBA LIDER 2" )
      wire#w1
      Contact( "AD5" )
      wire#w2
      Coil( "ARRANQUE BOMBA A" )
   END_RUNG
   RUNG wire#w1
      I_Contact( "DISPONIBLE BOMBA F" )
      Contact( "AD4" )
   END_RUNG wire#w2
   RUNG wire#powerrail
      Contact( "BOMBA LIDER 3" )
      wire#w3
      Contact( "AD4" )
   END_RUNG wire#w2
   RUNG wire#w3
      I_Contact( "DISPONIBLE BOMBA F" )
      Contact( "AD3" )
   END_RUNG wire#w2
   RUNG wire#powerrail
      Contact( "BOMBA LIDER 4" )
      wire#w4
      Contact( "AD3" )
   END_RUNG wire#w2
   RUNG wire#w4
      I_Contact( "DISPONIBLE BOMBA F" )
      Contact( "AD2" )
   END_RUNG wire#w2
   RUNG wire#powerrail
      Contact( "BOMBA LIDER 5" )
      wire#w5
      Contact( "AD2" )
   END_RUNG wire#w2
   RUNG wire#w5
      I_Contact( "DISPONIBLE BOMBA F" )
      Contact( "AD1" )
   END_RUNG wire#w2
   RUNG wire#powerrail
      Contact( "BOMBA LIDER 6" )
      Contact( "AD1" )
   END_RUNG wire#w2
   // the same network as SCL:
   "ARRANQUE BOMBA A" := ("BOMBA LIDER 2" AND ("AD5" OR (NOT "DISPONIBLE BOMBA F" AND "AD4"))) OR ("BOMBA LIDER 3" AND ("AD4" OR (NOT "DISPONIBLE BOMBA F" AND "AD3"))) OR ("BOMBA LIDER 4" AND ("AD3" OR (NOT "DISPONIBLE BOMBA F" AND "AD2"))) OR ("BOMBA LIDER 5" AND ("AD2" OR (NOT "DISPONIBLE BOMBA F" AND "AD1"))) OR ("BOMBA LIDER 6" AND "AD1");
END_REGION

REGION Network 22: ARRANQUE B2
   RUNG wire#powerrail
      Contact( "BOMBA LIDER 3" )
      wire#w1
      Contact( "AD5" )
      wire#w2
      Coil( "ARRANQUE BOMBA B" )
   END_RUNG
   RUNG wire#w1
      I_Contact( "DISPONIBLE BOMBA A" )
      Contact( "AD4" )
   END_RUNG wire#w2
   RUNG wire#powerrail
      Contact( "BOMBA LIDER 4" )
      wire#w3
      Contact( "AD4" )
   END_RUNG wire#w2
   RUNG wire#w3
      I_Contact( "DISPONIBLE BOMBA A" )
      Contact( "AD3" )
   END_RUNG wire#w2
   RUNG wire#powerrail
      Contact( "BOMBA LIDER 5" )
      wire#w4
      Contact( "AD3" )
   END_RUNG wire#w2
   RUNG wire#w4
      I_Contact( "DISPONIBLE BOMBA A" )
      Contact( "AD2" )
   END_RUNG wire#w2
   RUNG wire#powerrail
      Contact( "BOMBA LIDER 6" )
      wire#w5
      Contact( "AD2" )
   END_RUNG wire#w2
   RUNG wire#w5
      I_Contact( "DISPONIBLE BOMBA A" )
      Contact( "AD1" )
   END_RUNG wire#w2
   RUNG wire#powerrail
      Contact( "BOMBA LIDER 1" )
      Contact( "AD1" )
   END_RUNG wire#w2
   // the same network as SCL:
   "ARRANQUE BOMBA B" := ("BOMBA LIDER 3" AND ("AD5" OR (NOT "DISPONIBLE BOMBA A" AND "AD4"))) OR ("BOMBA LIDER 4" AND ("AD4" OR (NOT "DISPONIBLE BOMBA A" AND "AD3"))) OR ("BOMBA LIDER 5" AND ("AD3" OR (NOT "DISPONIBLE BOMBA A" AND "AD2"))) OR ("BOMBA LIDER 6" AND ("AD2" OR (NOT "DISPONIBLE BOMBA A" AND "AD1"))) OR ("BOMBA LIDER 1" AND "AD1");
END_REGION

REGION Network 23: ARRANQUE B3
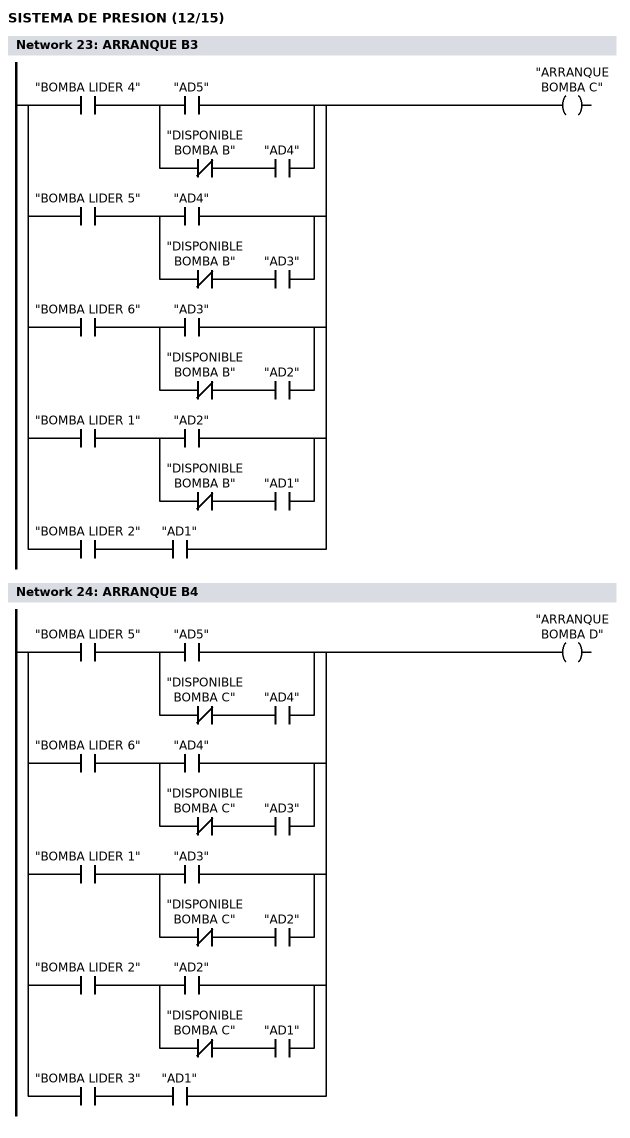
   RUNG wire#powerrail
      Contact( "BOMBA LIDER 4" )
      wire#w1
      Contact( "AD5" )
      wire#w2
      Coil( "ARRANQUE BOMBA C" )
   END_RUNG
   RUNG wire#w1
      I_Contact( "DISPONIBLE BOMBA B" )
      Contact( "AD4" )
   END_RUNG wire#w2
   RUNG wire#powerrail
      Contact( "BOMBA LIDER 5" )
      wire#w3
      Contact( "AD4" )
   END_RUNG wire#w2
   RUNG wire#w3
      I_Contact( "DISPONIBLE BOMBA B" )
      Contact( "AD3" )
   END_RUNG wire#w2
   RUNG wire#powerrail
      Contact( "BOMBA LIDER 6" )
      wire#w4
      Contact( "AD3" )
   END_RUNG wire#w2
   RUNG wire#w4
      I_Contact( "DISPONIBLE BOMBA B" )
      Contact( "AD2" )
   END_RUNG wire#w2
   RUNG wire#powerrail
      Contact( "BOMBA LIDER 1" )
      wire#w5
      Contact( "AD2" )
   END_RUNG wire#w2
   RUNG wire#w5
      I_Contact( "DISPONIBLE BOMBA B" )
      Contact( "AD1" )
   END_RUNG wire#w2
   RUNG wire#powerrail
      Contact( "BOMBA LIDER 2" )
      Contact( "AD1" )
   END_RUNG wire#w2
   // the same network as SCL:
   "ARRANQUE BOMBA C" := ("BOMBA LIDER 4" AND ("AD5" OR (NOT "DISPONIBLE BOMBA B" AND "AD4"))) OR ("BOMBA LIDER 5" AND ("AD4" OR (NOT "DISPONIBLE BOMBA B" AND "AD3"))) OR ("BOMBA LIDER 6" AND ("AD3" OR (NOT "DISPONIBLE BOMBA B" AND "AD2"))) OR ("BOMBA LIDER 1" AND ("AD2" OR (NOT "DISPONIBLE BOMBA B" AND "AD1"))) OR ("BOMBA LIDER 2" AND "AD1");
END_REGION

REGION Network 24: ARRANQUE B4
   RUNG wire#powerrail
      Contact( "BOMBA LIDER 5" )
      wire#w1
      Contact( "AD5" )
      wire#w2
      Coil( "ARRANQUE BOMBA D" )
   END_RUNG
   RUNG wire#w1
      I_Contact( "DISPONIBLE BOMBA C" )
      Contact( "AD4" )
   END_RUNG wire#w2
   RUNG wire#powerrail
      Contact( "BOMBA LIDER 6" )
      wire#w3
      Contact( "AD4" )
   END_RUNG wire#w2
   RUNG wire#w3
      I_Contact( "DISPONIBLE BOMBA C" )
      Contact( "AD3" )
   END_RUNG wire#w2
   RUNG wire#powerrail
      Contact( "BOMBA LIDER 1" )
      wire#w4
      Contact( "AD3" )
   END_RUNG wire#w2
   RUNG wire#w4
      I_Contact( "DISPONIBLE BOMBA C" )
      Contact( "AD2" )
   END_RUNG wire#w2
   RUNG wire#powerrail
      Contact( "BOMBA LIDER 2" )
      wire#w5
      Contact( "AD2" )
   END_RUNG wire#w2
   RUNG wire#w5
      I_Contact( "DISPONIBLE BOMBA C" )
      Contact( "AD1" )
   END_RUNG wire#w2
   RUNG wire#powerrail
      Contact( "BOMBA LIDER 3" )
      Contact( "AD1" )
   END_RUNG wire#w2
   // the same network as SCL:
   "ARRANQUE BOMBA D" := ("BOMBA LIDER 5" AND ("AD5" OR (NOT "DISPONIBLE BOMBA C" AND "AD4"))) OR ("BOMBA LIDER 6" AND ("AD4" OR (NOT "DISPONIBLE BOMBA C" AND "AD3"))) OR ("BOMBA LIDER 1" AND ("AD3" OR (NOT "DISPONIBLE BOMBA C" AND "AD2"))) OR ("BOMBA LIDER 2" AND ("AD2" OR (NOT "DISPONIBLE BOMBA C" AND "AD1"))) OR ("BOMBA LIDER 3" AND "AD1");
END_REGION

REGION Network 25: ARRANQUE B5
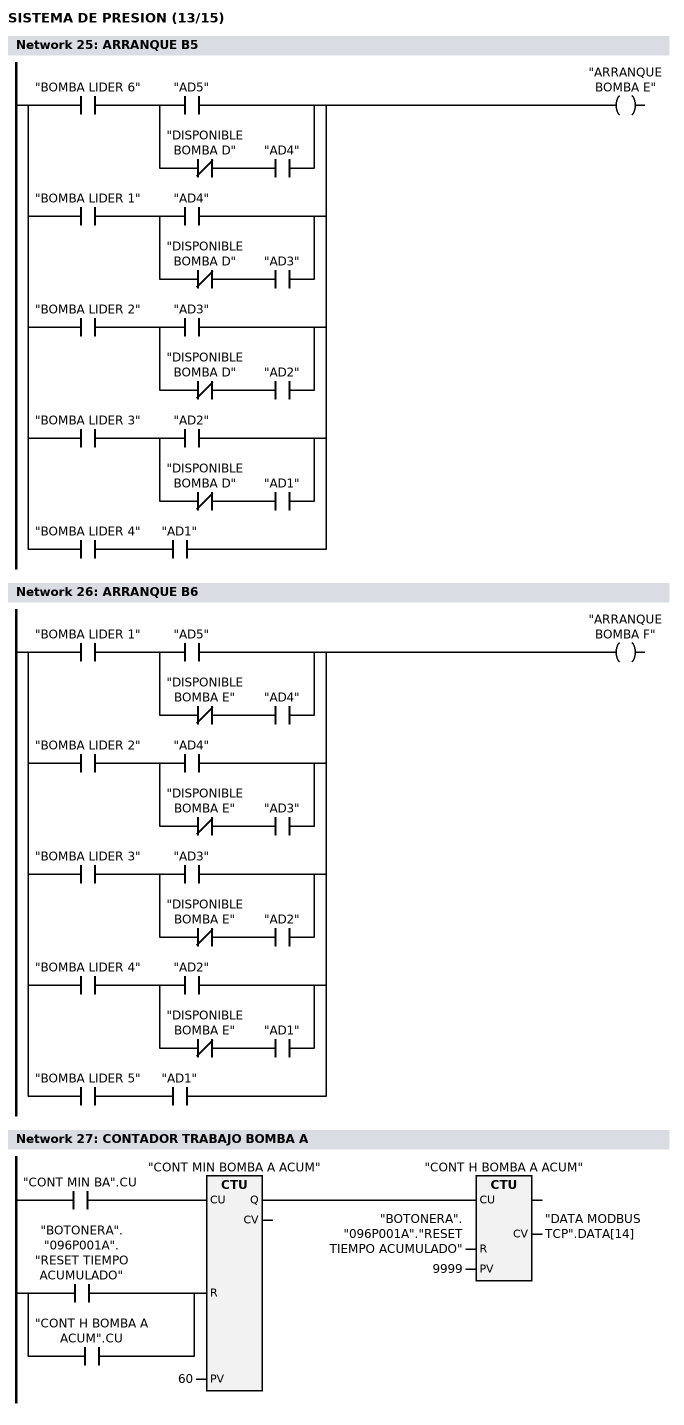
   RUNG wire#powerrail
      Contact( "BOMBA LIDER 6" )
      wire#w1
      Contact( "AD5" )
      wire#w2
      Coil( "ARRANQUE BOMBA E" )
   END_RUNG
   RUNG wire#w1
      I_Contact( "DISPONIBLE BOMBA D" )
      Contact( "AD4" )
   END_RUNG wire#w2
   RUNG wire#powerrail
      Contact( "BOMBA LIDER 1" )
      wire#w3
      Contact( "AD4" )
   END_RUNG wire#w2
   RUNG wire#w3
      I_Contact( "DISPONIBLE BOMBA D" )
      Contact( "AD3" )
   END_RUNG wire#w2
   RUNG wire#powerrail
      Contact( "BOMBA LIDER 2" )
      wire#w4
      Contact( "AD3" )
   END_RUNG wire#w2
   RUNG wire#w4
      I_Contact( "DISPONIBLE BOMBA D" )
      Contact( "AD2" )
   END_RUNG wire#w2
   RUNG wire#powerrail
      Contact( "BOMBA LIDER 3" )
      wire#w5
      Contact( "AD2" )
   END_RUNG wire#w2
   RUNG wire#w5
      I_Contact( "DISPONIBLE BOMBA D" )
      Contact( "AD1" )
   END_RUNG wire#w2
   RUNG wire#powerrail
      Contact( "BOMBA LIDER 4" )
      Contact( "AD1" )
   END_RUNG wire#w2
   // the same network as SCL:
   "ARRANQUE BOMBA E" := ("BOMBA LIDER 6" AND ("AD5" OR (NOT "DISPONIBLE BOMBA D" AND "AD4"))) OR ("BOMBA LIDER 1" AND ("AD4" OR (NOT "DISPONIBLE BOMBA D" AND "AD3"))) OR ("BOMBA LIDER 2" AND ("AD3" OR (NOT "DISPONIBLE BOMBA D" AND "AD2"))) OR ("BOMBA LIDER 3" AND ("AD2" OR (NOT "DISPONIBLE BOMBA D" AND "AD1"))) OR ("BOMBA LIDER 4" AND "AD1");
END_REGION

REGION Network 26: ARRANQUE B6
   RUNG wire#powerrail
      Contact( "BOMBA LIDER 1" )
      wire#w1
      Contact( "AD5" )
      wire#w2
      Coil( "ARRANQUE BOMBA F" )
   END_RUNG
   RUNG wire#w1
      I_Contact( "DISPONIBLE BOMBA E" )
      Contact( "AD4" )
   END_RUNG wire#w2
   RUNG wire#powerrail
      Contact( "BOMBA LIDER 2" )
      wire#w3
      Contact( "AD4" )
   END_RUNG wire#w2
   RUNG wire#w3
      I_Contact( "DISPONIBLE BOMBA E" )
      Contact( "AD3" )
   END_RUNG wire#w2
   RUNG wire#powerrail
      Contact( "BOMBA LIDER 3" )
      wire#w4
      Contact( "AD3" )
   END_RUNG wire#w2
   RUNG wire#w4
      I_Contact( "DISPONIBLE BOMBA E" )
      Contact( "AD2" )
   END_RUNG wire#w2
   RUNG wire#powerrail
      Contact( "BOMBA LIDER 4" )
      wire#w5
      Contact( "AD2" )
   END_RUNG wire#w2
   RUNG wire#w5
      I_Contact( "DISPONIBLE BOMBA E" )
      Contact( "AD1" )
   END_RUNG wire#w2
   RUNG wire#powerrail
      Contact( "BOMBA LIDER 5" )
      Contact( "AD1" )
   END_RUNG wire#w2
   // the same network as SCL:
   "ARRANQUE BOMBA F" := ("BOMBA LIDER 1" AND ("AD5" OR (NOT "DISPONIBLE BOMBA E" AND "AD4"))) OR ("BOMBA LIDER 2" AND ("AD4" OR (NOT "DISPONIBLE BOMBA E" AND "AD3"))) OR ("BOMBA LIDER 3" AND ("AD3" OR (NOT "DISPONIBLE BOMBA E" AND "AD2"))) OR ("BOMBA LIDER 4" AND ("AD2" OR (NOT "DISPONIBLE BOMBA E" AND "AD1"))) OR ("BOMBA LIDER 5" AND "AD1");
END_REGION

REGION Network 27: CONTADOR TRABAJO BOMBA A
   "CONT MIN BOMBA A ACUM".CTU(CU := "CONT MIN BA".CU,
                           R := "BOTONERA"."096P001A"."RESET TIEMPO ACUMULADO" OR "CONT H BOMBA A ACUM".CU,
                           PV := 60);
   "CONT H BOMBA A ACUM".CTU(CU := "CONT MIN BOMBA A ACUM".Q,
                           R := "BOTONERA"."096P001A"."RESET TIEMPO ACUMULADO",
                           PV := 9999,
                           CV => "DATA MODBUS TCP".DATA[14]);
END_REGION

REGION Network 28: CONTADOR TRABAJO BOMBA B
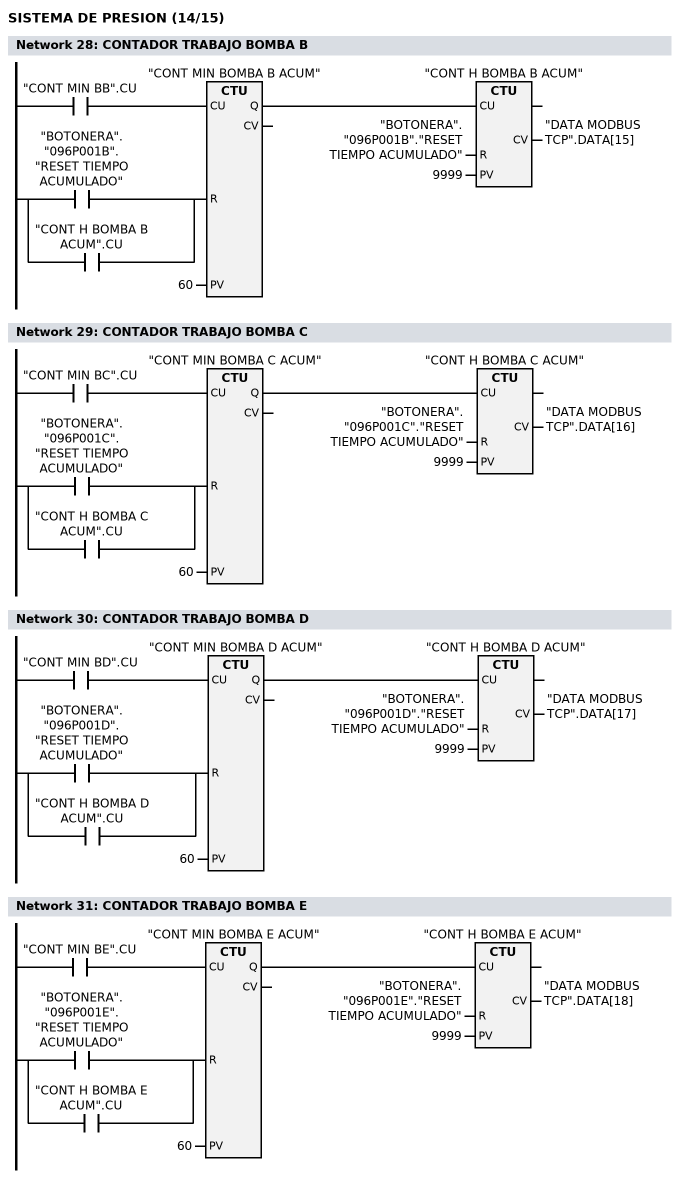
   "CONT MIN BOMBA B ACUM".CTU(CU := "CONT MIN BB".CU,
                           R := "BOTONERA"."096P001B"."RESET TIEMPO ACUMULADO" OR "CONT H BOMBA B ACUM".CU,
                           PV := 60);
   "CONT H BOMBA B ACUM".CTU(CU := "CONT MIN BOMBA B ACUM".Q,
                           R := "BOTONERA"."096P001B"."RESET TIEMPO ACUMULADO",
                           PV := 9999,
                           CV => "DATA MODBUS TCP".DATA[15]);
END_REGION

REGION Network 29: CONTADOR TRABAJO BOMBA C
   "CONT MIN BOMBA C ACUM".CTU(CU := "CONT MIN BC".CU,
                           R := "BOTONERA"."096P001C"."RESET TIEMPO ACUMULADO" OR "CONT H BOMBA C ACUM".CU,
                           PV := 60);
   "CONT H BOMBA C ACUM".CTU(CU := "CONT MIN BOMBA C ACUM".Q,
                           R := "BOTONERA"."096P001C"."RESET TIEMPO ACUMULADO",
                           PV := 9999,
                           CV => "DATA MODBUS TCP".DATA[16]);
END_REGION

REGION Network 30: CONTADOR TRABAJO BOMBA D
   "CONT MIN BOMBA D ACUM".CTU(CU := "CONT MIN BD".CU,
                           R := "BOTONERA"."096P001D"."RESET TIEMPO ACUMULADO" OR "CONT H BOMBA D ACUM".CU,
                           PV := 60);
   "CONT H BOMBA D ACUM".CTU(CU := "CONT MIN BOMBA D ACUM".Q,
                           R := "BOTONERA"."096P001D"."RESET TIEMPO ACUMULADO",
                           PV := 9999,
                           CV => "DATA MODBUS TCP".DATA[17]);
END_REGION

REGION Network 31: CONTADOR TRABAJO BOMBA E
   "CONT MIN BOMBA E ACUM".CTU(CU := "CONT MIN BE".CU,
                           R := "BOTONERA"."096P001E"."RESET TIEMPO ACUMULADO" OR "CONT H BOMBA E ACUM".CU,
                           PV := 60);
   "CONT H BOMBA E ACUM".CTU(CU := "CONT MIN BOMBA E ACUM".Q,
                           R := "BOTONERA"."096P001E"."RESET TIEMPO ACUMULADO",
                           PV := 9999,
                           CV => "DATA MODBUS TCP".DATA[18]);
END_REGION

REGION Network 32: CONTADOR TRABAJO BOMBA F
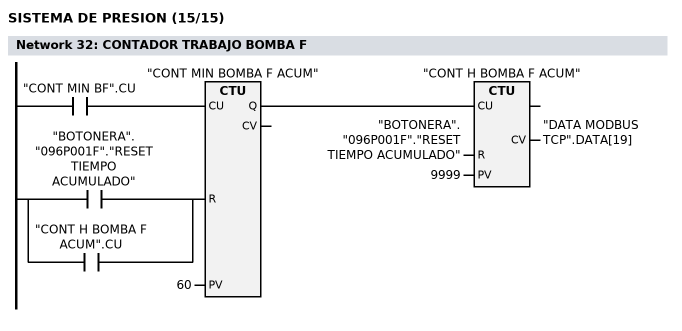
   "CONT MIN BOMBA F ACUM".CTU(CU := "CONT MIN BF".CU,
                           R := "BOTONERA"."096P001F"."RESET TIEMPO ACUMULADO" OR "CONT H BOMBA F ACUM".CU,
                           PV := 60);
   "CONT H BOMBA F ACUM".CTU(CU := "CONT MIN BOMBA F ACUM".Q,
                           R := "BOTONERA"."096P001F"."RESET TIEMPO ACUMULADO",
                           PV := 9999,
                           CV => "DATA MODBUS TCP".DATA[19]);
END_REGION
END_FUNCTION

FUNCTION "Comunicacion RTU" : Void   // FC5, LAD
{ S7_Optimized_Access := 'TRUE' }
VERSION : 0.1
   VAR_TEMP
      "RESET TEMP" : Bool;
      TEST1 : Bool;
      error1 : Bool;
      error2 : Bool;
      error3 : Bool;
      error4 : Bool;
      error5 : Bool;
      error6 : Bool;
      error7 : Bool;
      error8 : Bool;
      error9 : Bool;
      error10 : Bool;
      error11 : Bool;
      error12 : Bool;
      error13 : Bool;
      error14 : Bool;
      error15 : Bool;
      error16 : Bool;
      error17 : Bool;
      error18 : Bool;
      error19 : Bool;
      error20 : Bool;
      error21 : Bool;
      error22 : Bool;
      error23 : Bool;
      error24 : Bool;
      error25 : Bool;
   END_VAR
BEGIN

REGION Network 1: CONTEO COMUNICACION
